FUNCTION "Sheet 4 (RSM)" : VOID	// FC 26
TITLE = Sheet 4 (RSM)
//HP FILM & TICM & TMAX (Analog)
AUTHOR : RJ
FAMILY : RSM
VERSION : 0.1
BEGIN
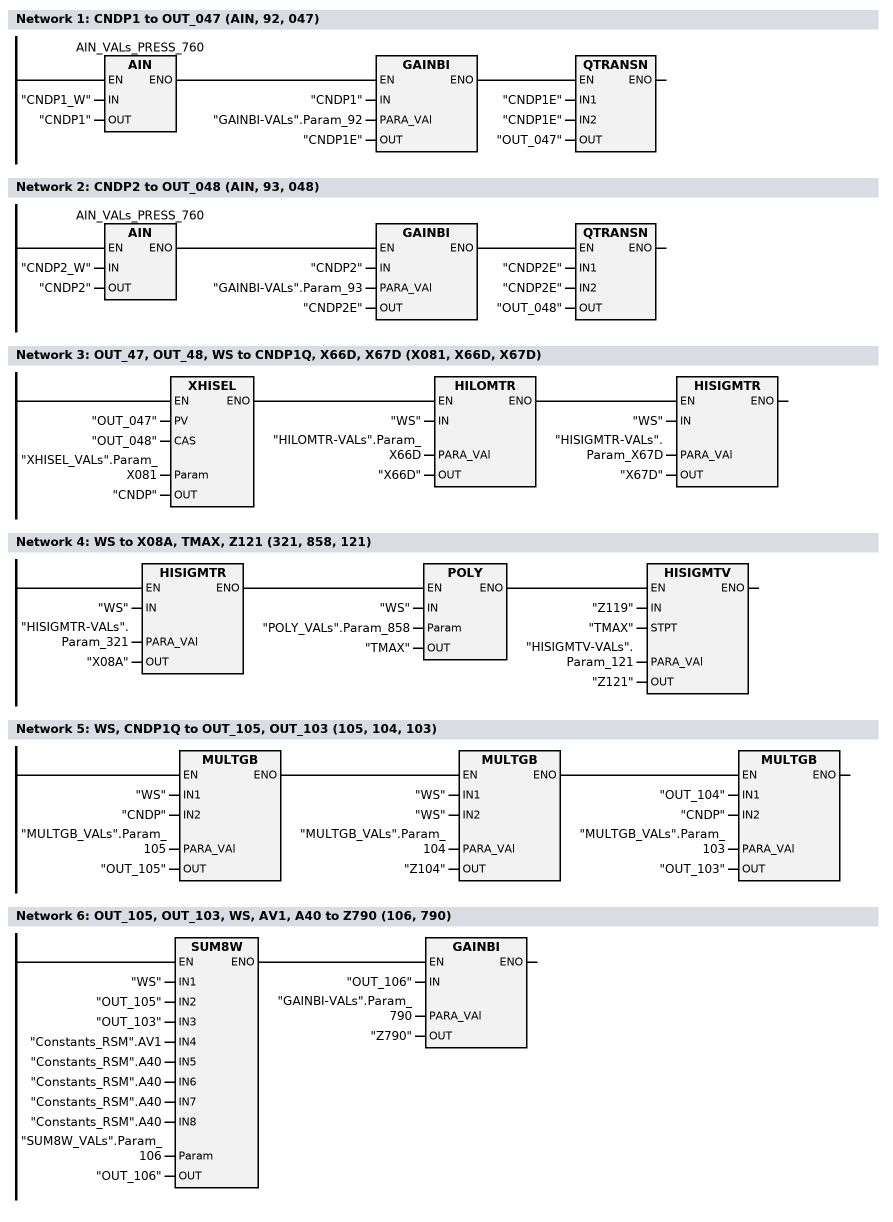
NETWORK
TITLE = CNDP1 to OUT_047 (AIN, 92, 047)
      A(;
      A(;
      CALL  "AIN" , "AIN_VALs_PRESS_760" (
           IN                       := "CNDP1_W",
           OUT                      := "CNDP1");
      A     BR;
      );
      JNB   _001;
      CALL  "GAINBI" (
           IN                       := "CNDP1",
           PARA_VAl                 := "GAINBI-VALs".Param_92,
           OUT                      := "CNDP1E");
_001: A     BR;
      );
      JNB   _002;
      CALL  "QTRANSN" (
           IN1                      := "CNDP1E",
           IN2                      := "CNDP1E",
           OUT                      := "OUT_047");
_002: NOP   0;
NETWORK
TITLE = CNDP2 to OUT_048 (AIN, 93, 048)
      A(;
      A(;
      CALL  "AIN" , "AIN_VALs_PRESS_760" (
           IN                       := "CNDP2_W",
           OUT                      := "CNDP2");
      A     BR;
      );
      JNB   _003;
      CALL  "GAINBI" (
           IN                       := "CNDP2",
           PARA_VAl                 := "GAINBI-VALs".Param_93,
           OUT                      := "CNDP2E");
_003: A     BR;
      );
      JNB   _004;
      CALL  "QTRANSN" (
           IN1                      := "CNDP2E",
           IN2                      := "CNDP2E",
           OUT                      := "OUT_048");
_004: NOP   0;
NETWORK
TITLE = OUT_47, OUT_48, WS to CNDP1Q, X66D, X67D (X081, X66D, X67D)
      A(;
      A(;
      CALL  "XHISEL" (
           PV                       := "OUT_047",
           CAS                      := "OUT_048",
           Param                    := "XHISEL_VALs".Param_X081,
           OUT                      := "CNDP");
      A     BR;
      );
      JNB   _005;
      CALL  "HILOMTR" (
           IN                       := "WS",
           PARA_VAl                 := "HILOMTR-VALs".Param_X66D,
           OUT                      := "X66D");
_005: A     BR;
      );
      JNB   _006;
      CALL  "HISIGMTR" (
           IN                       := "WS",
           PARA_VAl                 := "HISIGMTR-VALs".Param_X67D,
           OUT                      := "X67D");
_006: NOP   0;
NETWORK
TITLE = WS to X08A, TMAX, Z121 (321, 858, 121)
      A(;
      A(;
      CALL  "HISIGMTR" (
           IN                       := "WS",
           PARA_VAl                 := "HISIGMTR-VALs".Param_321,
           OUT                      := "X08A");
      A     BR;
      );
      JNB   _007;
      CALL  "POLY" (
           IN                       := "WS",
           Param                    := "POLY_VALs".Param_858,
           OUT                      := "TMAX");
_007: A     BR;
      );
      JNB   _008;
      CALL  "HISIGMTV" (
           IN                       := "Z119",
           STPT                     := "TMAX",
           PARA_VAl                 := "HISIGMTV-VALs".Param_121,
           OUT                      := "Z121");
_008: NOP   0;
NETWORK
TITLE = WS, CNDP1Q to OUT_105, OUT_103 (105, 104, 103)
      A(;
      A(;
      CALL  "MULTGB" (
           IN1                      := "WS",
           IN2                      := "CNDP",
           PARA_VAl                 := "MULTGB_VALs".Param_105,
           OUT                      := "OUT_105");
      A     BR;
      );
      JNB   _009;
      CALL  "MULTGB" (
           IN1                      := "WS",
           IN2                      := "WS",
           PARA_VAl                 := "MULTGB_VALs".Param_104,
           OUT                      := "Z104");
_009: A     BR;
      );
      JNB   _00a;
      CALL  "MULTGB" (
           IN1                      := "OUT_104",
           IN2                      := "CNDP",
           PARA_VAl                 := "MULTGB_VALs".Param_103,
           OUT                      := "OUT_103");
_00a: NOP   0;
NETWORK
TITLE = OUT_105, OUT_103, WS, AV1, A40 to Z790 (106, 790)
      A(;
      CALL  "SUM8W" (
           IN1                      := "WS",
           IN2                      := "OUT_105",
           IN3                      := "OUT_103",
           IN4                      := "Constants_RSM".AV1,
           IN5                      := "Constants_RSM".A40,
           IN6                      := "Constants_RSM".A40,
           IN7                      := "Constants_RSM".A40,
           IN8                      := "Constants_RSM".A40,
           Param                    := "SUM8W_VALs".Param_106,
           OUT                      := "OUT_106");
      A     BR;
      );
      JNB   _00b;
      CALL  "GAINBI" (
           IN                       := "OUT_106",
           PARA_VAl                 := "GAINBI-VALs".Param_790,
           OUT                      := "Z790");
_00b: NOP   0;
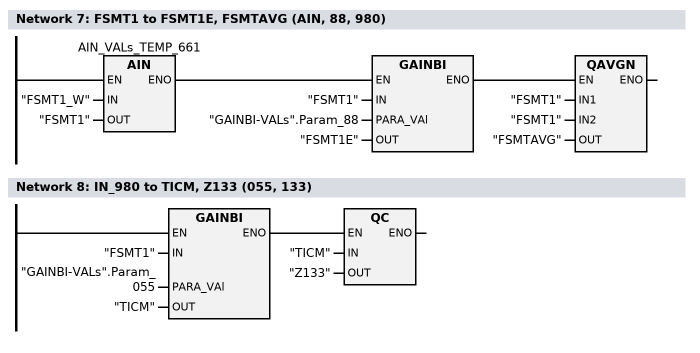
NETWORK
TITLE = FSMT1 to FSMT1E, FSMTAVG (AIN, 88, 980)
      A(;
      A(;
      CALL  "AIN" , "AIN_VALs_TEMP_661" (
           IN                       := "FSMT1_W",
           OUT                      := "FSMT1");
      A     BR;
      );
      JNB   _00c;
      CALL  "GAINBI" (
           IN                       := "FSMT1",
           PARA_VAl                 := "GAINBI-VALs".Param_88,
           OUT                      := "FSMT1E");
_00c: A     BR;
      );
      JNB   _00d;
      CALL  "QAVGN" (
           IN1                      := "FSMT1",
           IN2                      := "FSMT1",
           OUT                      := "FSMTAVG");
_00d: NOP   0;
NETWORK
TITLE = IN_980 to TICM, Z133 (055, 133)
      A(;
      CALL  "GAINBI" (
           IN                       := "FSMT1",
           PARA_VAl                 := "GAINBI-VALs".Param_055,
           OUT                      := "TICM");
      A     BR;
      );
      JNB   _00e;
      CALL  "QC" (
           IN                       := "TICM",
           OUT                      := "Z133");
_00e: NOP   0;
END_FUNCTION

FUNCTION "Sheet 5 (RSM)" : VOID	// FC 27
TITLE = Sheet 5 (RSM)
//MWINC LOGIC (Digital)
AUTHOR : RJ
FAMILY : RSM
VERSION : 0.1
BEGIN
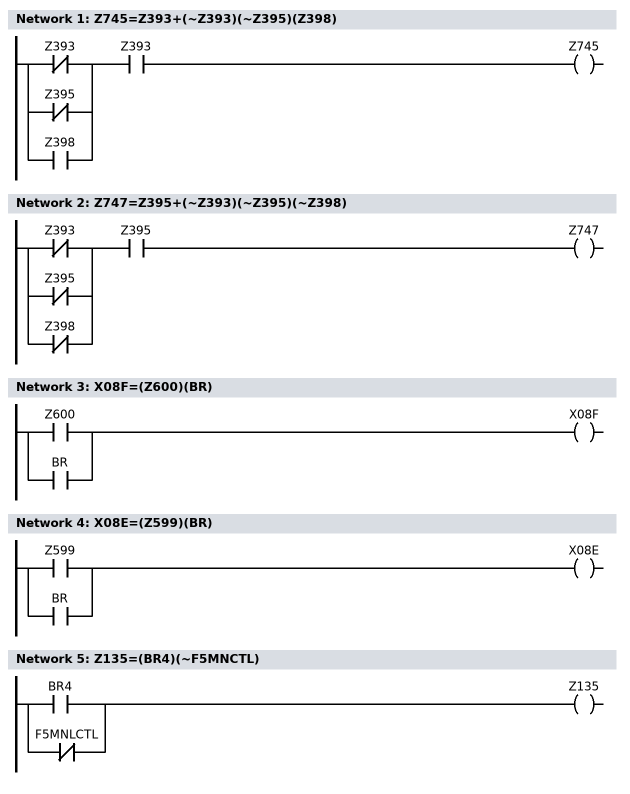
NETWORK
TITLE = Z745=Z393+(~Z393)(~Z395)(Z398)
      A(;
      ON    "Z393";
      ON    "Z395";
      O     "Z398";
      );
      A     "Z393";
      =     "Z745";
NETWORK
TITLE = Z747=Z395+(~Z393)(~Z395)(~Z398)
      A(;
      ON    "Z393";
      ON    "Z395";
      ON    "Z398";
      );
      A     "Z395";
      =     "Z747";
NETWORK
TITLE = X08F=(Z600)(BR)
      O     "Z600";
      O     "BR";
      =     "X08F";
NETWORK
TITLE = X08E=(Z599)(BR)
      O     "Z599";
      O     "BR";
      =     "X08E";
NETWORK
TITLE = Z135=(BR4)(~F5MNCTL)
      O     "BR4";
      ON    "F5MNLCTL";
      =     "Z135";
END_FUNCTION

FUNCTION "Sheet 7 (RSM)" : VOID	// FC 28
TITLE = Sheet 7 (RSM)
//HP INVALID LOGIC (Digital)
//
AUTHOR : RJ
FAMILY : RSM
VERSION : 0.1
BEGIN
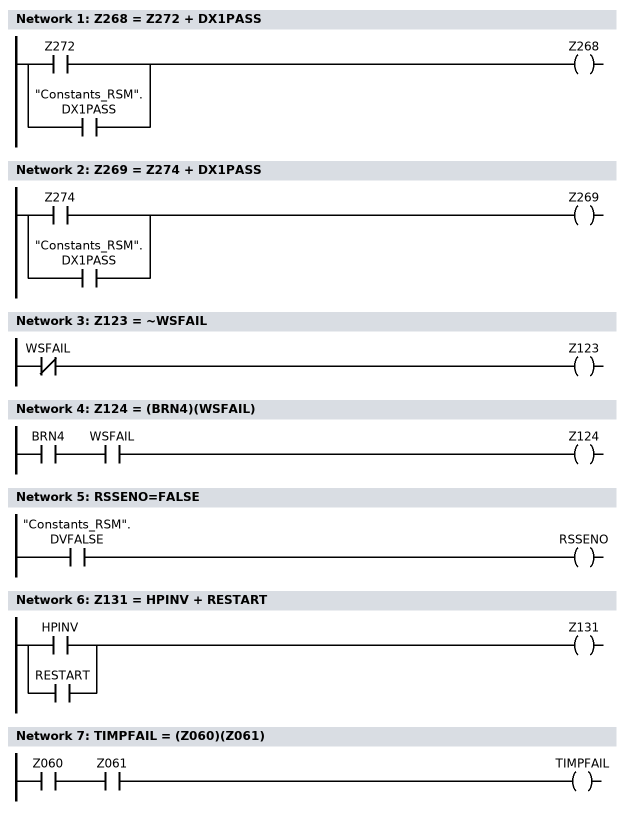
NETWORK
TITLE = Z268 = Z272 + DX1PASS
      O     "Z272";
      O     "Constants_RSM".DX1PASS;
      =     "Z268";
NETWORK
TITLE = Z269 = Z274 + DX1PASS
      O     "Z274";
      O     "Constants_RSM".DX1PASS;
      =     "Z269";
NETWORK
TITLE = Z123 = ~WSFAIL
      AN    "WSFAIL";
      =     "Z123";
NETWORK
TITLE = Z124 = (BRN4)(WSFAIL)
      A     "BRN4";
      A     "WSFAIL";
      =     "Z124";
NETWORK
TITLE = RSSENO=FALSE
      A     "Constants_RSM".DVFALSE;
      =     "RSSENO";
NETWORK
TITLE = Z131 = HPINV + RESTART
      O     "HPINV";
      O     "RESTART";
      =     "Z131";
NETWORK
TITLE = TIMPFAIL = (Z060)(Z061)
      A     "Z060";
      A     "Z061";
      =     "TIMPFAIL";
NETWORK
TITLE = RESTART Singnal logic
//RESTART=RTRSWSFL+DVFALSE+TIMPFAIL+(RESTART)(Z133)+(DX1PASS)(OUT_180)
      O     "RTRSWSFL";
      O     "Constants_RSM".DVFALSE;
      O     "TIMPFAIL";
      O;
      A     "Z133";
      A     "RESTART";
      O(;
      A     "Constants_RSM".DX1PASS;
      S     "OUT_180";
      A     "OUT_180";
      R     "OUT_180";
      A     "OUT_180";
      );
      =     "RESTART";
END_FUNCTION

FUNCTION "RESETSUM" : VOID	// FC 29
AUTHOR : RJ
VERSION : 0.0
VAR_INPUT
  FFLG : BOOL ;
  RSET : BOOL ;
  RUN : BOOL ;
  IN : REAL ;
  Param : STRUCT
   RCNT : REAL ;
   GAIN : REAL ;
   TRST : REAL ;
  END_STRUCT ;
END_VAR
VAR_IN_OUT
  OUT : REAL ;
END_VAR
VAR_TEMP
  TEMP : REAL ;
  RCNT : REAL ;
  GAIN : REAL ;
  TRST : REAL ;
END_VAR
BEGIN
// body was compiled from an SCL source; compiled code not shown
END_FUNCTION

FUNCTION "Sheet 6 (RSM)" : VOID	// FC 30
TITLE = Sheet 6 (RSM)
//HP Stress Counters (Analog)
AUTHOR : RJ
FAMILY : RSM
VERSION : 0.1
BEGIN
NETWORK
TITLE = AV1, DVFALSE, RESTART to X080, HPINV, HPICOL (129, 320, 130)
      A(;
      A(;
      A     "Constants_RSM".DVFALSE;
      =     L 0.0;
      BLD   103;
      A     "RESTART";
      =     L 0.1;
      BLD   103;
      A     "Z131";
      =     L 0.2;
      BLD   103;
      CALL  "RESETSUM" (
           FFLG                     := L 0.0,
           RSET                     := L 0.1,
           RUN                      := L 0.2,
           IN                       := "Constants_RSM".AV1,
           Param                    := "RESETSUM_VALs".Param_129,
           OUT                      := "HPICOL");
      A     BR;
      );
      JNB   _001;
      CALL  "HISIGMTR" (
           IN                       := "HPICOL",
           PARA_VAl                 := "HISIGMTR-VALs".Param_320,
           OUT                      := "X08D");
_001: A     BR;
      );
      JNB   _002;
      CALL  "LOSIGMTR" (
           IN                       := "HPICOL",
           PARA_VAl                 := "LOSIGMTR-VALs".Param_130,
           OUT                      := "HPINV");
_002: NOP   0;
NETWORK
TITLE = AV1, HPICOL to Z272 (270, 271, 272)
      A(;
      A     "Constants_RSM".DVFALSE;
      =     L 0.0;
      BLD   103;
      A     "Z272";
      =     L 0.1;
      BLD   103;
      A     "OUT_270";
      =     L 0.2;
      BLD   103;
      A(;
      CALL  "HISIGMTR" (
           IN                       := "HPICOL",
           PARA_VAl                 := "HISIGMTR-VALs".Param_270,
           OUT                      := "OUT_270");
      A     BR;
      );
      JNB   _003;
      CALL  "RESETSUM" (
           FFLG                     := L 0.0,
           RSET                     := L 0.1,
           RUN                      := L 0.2,
           IN                       := "Constants_RSM".AV1,
           Param                    := "RESETSUM_VALs".Param_271,
           OUT                      := "ONEMINCT");
_003: A     BR;
      );
      JNB   _004;
      CALL  "HISIGMTR" (
           IN                       := "ONEMINCT",
           PARA_VAl                 := "HISIGMTR-VALs".Param_272,
           OUT                      := "Z272");
_004: NOP   0;
NETWORK
TITLE = AV1, DVFALSE, DVTRUE to T5SEC (317, 318)
      A(;
      A     "Constants_RSM".DVFALSE;
      =     L 0.0;
      BLD   103;
      A     "T5SEC";
      =     L 0.1;
      BLD   103;
      A     "Constants_RSM".DVTRUE;
      =     L 0.2;
      BLD   103;
      CALL  "RESETSUM" (
           FFLG                     := L 0.0,
           RSET                     := L 0.1,
           RUN                      := L 0.2,
           IN                       := "Constants_RSM".AV1,
           Param                    := "RESETSUM_VALs".Param_317,
           OUT                      := "OUT_317");
      A     BR;
      );
      JNB   _005;
      CALL  "HISIGMTR" (
           IN                       := "OUT_317",
           PARA_VAl                 := "HISIGMTR-VALs".Param_318,
           OUT                      := "T5SEC");
_005: NOP   0;
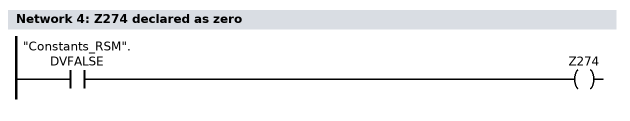
NETWORK
TITLE = Z274 declared as zero
      A     "Constants_RSM".DVFALSE;
      =     "Z274";
NETWORK
TITLE = AV1, Z123, Z124 to RTRSWSFL (125, 126)
      A(;
      A     "Constants_RSM".DVFALSE;
      =     L 0.0;
      BLD   103;
      A     "Z123";
      =     L 0.1;
      BLD   103;
      A     "Z124";
      =     L 0.2;
      BLD   103;
      CALL  "RESETSUM" (
           FFLG                     := L 0.0,
           RSET                     := L 0.1,
           RUN                      := L 0.2,
           IN                       := "Constants_RSM".AV1,
           Param                    := "RESETSUM_VALs".Param_136,
           OUT                      := "ISPOUTCT");
      A     BR;
      );
      JNB   _006;
      CALL  "HISIGMTR" (
           IN                       := "ISPOUTCT",
           PARA_VAl                 := "HISIGMTR-VALs".Param_137,
           OUT                      := "RTRSWSFL");
_006: NOP   0;
END_FUNCTION

FUNCTION "HISIGMTV" : VOID	// FC 31
AUTHOR : Sabeeh
VERSION : 0.0
VAR_INPUT
  IN : REAL ;
  STPT : REAL ;
  PARA_VAl : STRUCT
   DBAN : REAL ;
  END_STRUCT ;
END_VAR
VAR_OUTPUT
  OUT : BOOL ;
END_VAR
BEGIN
// body was compiled from an SCL source; compiled code not shown
END_FUNCTION

FUNCTION "LOSIGMTV" : VOID	// FC 32
AUTHOR : Sabeeh
VERSION : 0.0
VAR_INPUT
  IN1 : REAL ;
  STPT : REAL ;
  PARA_VAl : STRUCT
   DBAN : REAL ;
  END_STRUCT ;
END_VAR
VAR_OUTPUT
  FLAG : BOOL ;
END_VAR
BEGIN
// body was compiled from an SCL source; compiled code not shown
END_FUNCTION

FUNCTION "HISEL10" : VOID	// FC 33
AUTHOR : Sabeeh
VERSION : 0.0
VAR_INPUT
  IN1 : REAL ;
  IN2 : REAL ;
END_VAR
VAR_OUTPUT
  OUT : REAL ;
END_VAR
BEGIN
// body was compiled from an SCL source; compiled code not shown
END_FUNCTION

FUNCTION "XLIMIT" : VOID	// FC 34
AUTHOR : Sabeeh
VERSION : 0.0
VAR_INPUT
  CAS : REAL ;
  PARA_VAl : STRUCT
   GAIN : REAL  := 1.000000e+000;
   BIAS : REAL ;
   SCLTOP : REAL  := 1.000000e+002;
   SCLBTM : REAL  := -1.000000e+002;
  END_STRUCT ;
END_VAR
VAR_OUTPUT
  OUT : REAL ;
END_VAR
VAR_TEMP
  TEMP : REAL ;
END_VAR
BEGIN
// body was compiled from an SCL source; compiled code not shown
END_FUNCTION

FUNCTION "LOSEL10" : VOID	// FC 35
AUTHOR : Sabeeh
VERSION : 0.0
VAR_INPUT
  IN1 : REAL ;
  IN2 : REAL ;
END_VAR
VAR_OUTPUT
  OUT : REAL ;
END_VAR
BEGIN
// body was compiled from an SCL source; compiled code not shown
END_FUNCTION

FUNCTION "Sheet 9 (RSM)" : VOID	// FC 36
TITLE = Sheet 9 (RSM)
//HP ROTSURF, T1-5 & TP1-4 (Analog)
AUTHOR : RJ
FAMILY : RSM
VERSION : 0.1
BEGIN
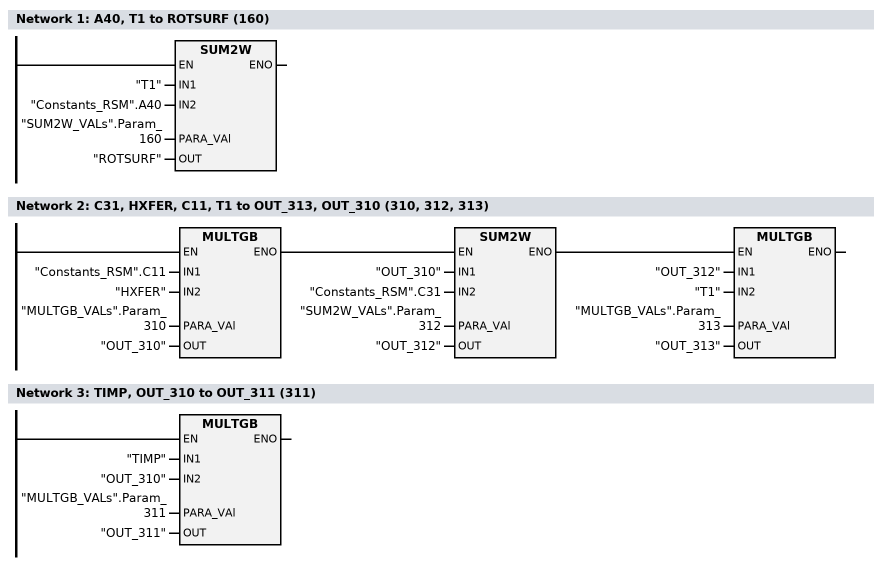
NETWORK
TITLE = A40, T1 to ROTSURF (160)
      CALL  "SUM2W" (
           IN1                      := "T1",
           IN2                      := "Constants_RSM".A40,
           PARA_VAl                 := "SUM2W_VALs".Param_160,
           OUT                      := "ROTSURF");
      NOP   0;
NETWORK
TITLE = C31, HXFER, C11, T1 to OUT_313, OUT_310 (310, 312, 313)
//IN1 of Block 312 should have a -ve weight w.r.f sheet 9 (RSM).
      A(;
      A(;
      CALL  "MULTGB" (
           IN1                      := "Constants_RSM".C11,
           IN2                      := "HXFER",
           PARA_VAl                 := "MULTGB_VALs".Param_310,
           OUT                      := "OUT_310");
      A     BR;
      );
      JNB   _001;
      CALL  "SUM2W" (
           IN1                      := "OUT_310",
           IN2                      := "Constants_RSM".C31,
           PARA_VAl                 := "SUM2W_VALs".Param_312,
           OUT                      := "OUT_312");
_001: A     BR;
      );
      JNB   _002;
      CALL  "MULTGB" (
           IN1                      := "OUT_312",
           IN2                      := "T1",
           PARA_VAl                 := "MULTGB_VALs".Param_313,
           OUT                      := "OUT_313");
_002: NOP   0;
NETWORK
TITLE = TIMP, OUT_310 to OUT_311 (311)
      CALL  "MULTGB" (
           IN1                      := "TIMP",
           IN2                      := "OUT_310",
           PARA_VAl                 := "MULTGB_VALs".Param_311,
           OUT                      := "OUT_311");
      NOP   0;
NETWORK
TITLE = Blocks 314, 315, 316
      A     "RESTART";
      =     L 0.0;
      BLD   103;
      A(;
      A     "T5SEC";
      =     L 0.1;
      BLD   103;
      A(;
      CALL  "SUM4W" (
           IN1                      := "OUT_311",
           IN2                      := "OUT_313",
           IN3                      := "T2",
           IN4                      := "Constants_RSM".A40,
           PARA_VAl                 := "SUM4W_VALs".Param_314,
           OUT                      := "TP1");
      A     BR;
      );
      JNB   _003;
      CALL  "TRANSF" (
           FLAG                     := L 0.1,
           IN1_y                    := "TP1",
           IN2_n                    := "T1",
           OUT                      := "OUT_315");
_003: A     BR;
      );
      JNB   _004;
      CALL  "TRANSF" (
           FLAG                     := L 0.0,
           IN1_y                    := "TICM",
           IN2_n                    := "OUT_315",
           OUT                      := "T1");
_004: NOP   0;
NETWORK
TITLE = Block 326, 327, 328
      A     "RESTART";
      =     L 0.0;
      BLD   103;
      A(;
      A     "T5SEC";
      =     L 0.1;
      BLD   103;
      A(;
      CALL  "SUM4W" (
           IN1                      := "T1",
           IN2                      := "T2",
           IN3                      := "T3",
           IN4                      := "Constants_RSM".A40,
           PARA_VAl                 := "SUM4W_VALs".Param_326,
           OUT                      := "TP2");
      A     BR;
      );
      JNB   _005;
      CALL  "TRANSF" (
           FLAG                     := L 0.1,
           IN1_y                    := "TP2",
           IN2_n                    := "T2",
           OUT                      := "OUT_327");
_005: A     BR;
      );
      JNB   _006;
      CALL  "TRANSF" (
           FLAG                     := L 0.0,
           IN1_y                    := "TICM",
           IN2_n                    := "OUT_327",
           OUT                      := "T2");
_006: NOP   0;
NETWORK
TITLE = Blocks 329, 330, 331
      A     "RESTART";
      =     L 0.0;
      BLD   103;
      A(;
      A     "T5SEC";
      =     L 0.1;
      BLD   103;
      A(;
      CALL  "SUM4W" (
           IN1                      := "T2",
           IN2                      := "T3",
           IN3                      := "T4",
           IN4                      := "Constants_RSM".A40,
           PARA_VAl                 := "SUM4W_VALs".Param_329,
           OUT                      := "TP3");
      A     BR;
      );
      JNB   _007;
      CALL  "TRANSF" (
           FLAG                     := L 0.1,
           IN1_y                    := "TP3",
           IN2_n                    := "T3",
           OUT                      := "OUT_330");
_007: A     BR;
      );
      JNB   _008;
      CALL  "TRANSF" (
           FLAG                     := L 0.0,
           IN1_y                    := "TICM",
           IN2_n                    := "OUT_330",
           OUT                      := "T3");
_008: NOP   0;
NETWORK
TITLE = Blocks 332, 333, 334
      A     "RESTART";
      =     L 0.0;
      BLD   103;
      A(;
      A     "T5SEC";
      =     L 0.1;
      BLD   103;
      A(;
      CALL  "SUM4W" (
           IN1                      := "T3",
           IN2                      := "T4",
           IN3                      := "T5",
           IN4                      := "Constants_RSM".A40,
           PARA_VAl                 := "SUM4W_VALs".Param_332,
           OUT                      := "TP4");
      A     BR;
      );
      JNB   _009;
      CALL  "TRANSF" (
           FLAG                     := L 0.1,
           IN1_y                    := "TP4",
           IN2_n                    := "T4",
           OUT                      := "OUT_333");
_009: A     BR;
      );
      JNB   _00a;
      CALL  "TRANSF" (
           FLAG                     := L 0.0,
           IN1_y                    := "TICM",
           IN2_n                    := "OUT_333",
           OUT                      := "T4");
_00a: NOP   0;
NETWORK
TITLE = Blocks 335, 336, 337
      A     "RESTART";
      =     L 0.0;
      BLD   103;
      A(;
      A     "T5SEC";
      =     L 0.1;
      BLD   103;
      A(;
      CALL  "SUM4W" (
           IN1                      := "T4",
           IN2                      := "T5",
           IN3                      := "T6",
           IN4                      := "Constants_RSM".A40,
           PARA_VAl                 := "SUM4W_VALs".Param_335,
           OUT                      := "TP5");
      A     BR;
      );
      JNB   _00b;
      CALL  "TRANSF" (
           FLAG                     := L 0.1,
           IN1_y                    := "TP5",
           IN2_n                    := "T5",
           OUT                      := "OUT_336");
_00b: A     BR;
      );
      JNB   _00c;
      CALL  "TRANSF" (
           FLAG                     := L 0.0,
           IN1_y                    := "TICM",
           IN2_n                    := "OUT_336",
           OUT                      := "T5");
_00c: NOP   0;
END_FUNCTION

FUNCTION "Sheet 8 (RSM)" : VOID	// FC 37
TITLE = Sheet 8 (RSM)
//HXFER & TWC (Analog)
AUTHOR : RJ
FAMILY : RSM
VERSION : 0.1
BEGIN
NETWORK
TITLE = Blocks 136, 137
      A(;
      A     "Constants_RSM".DVFALSE;
      =     L 0.0;
      BLD   103;
      A     "BRN4";
      =     L 0.1;
      BLD   103;
      A     "Z135";
      =     L 0.2;
      BLD   103;
      CALL  "RESETSUM" (
           FFLG                     := L 0.0,
           RSET                     := L 0.1,
           RUN                      := L 0.2,
           IN                       := "Constants_RSM".AV1,
           Param                    := P#DB30.DBX 60.0,
           OUT                      := "OUT_136");
      A     BR;
      );
      JNB   _001;
      CALL  "HISIGMTR" (
           IN                       := "OUT_136",
           PARA_VAl                 := "HISIGMTR-VALs".Param_221,
           OUT                      := "F5MNLCTL");
_001: NOP   0;
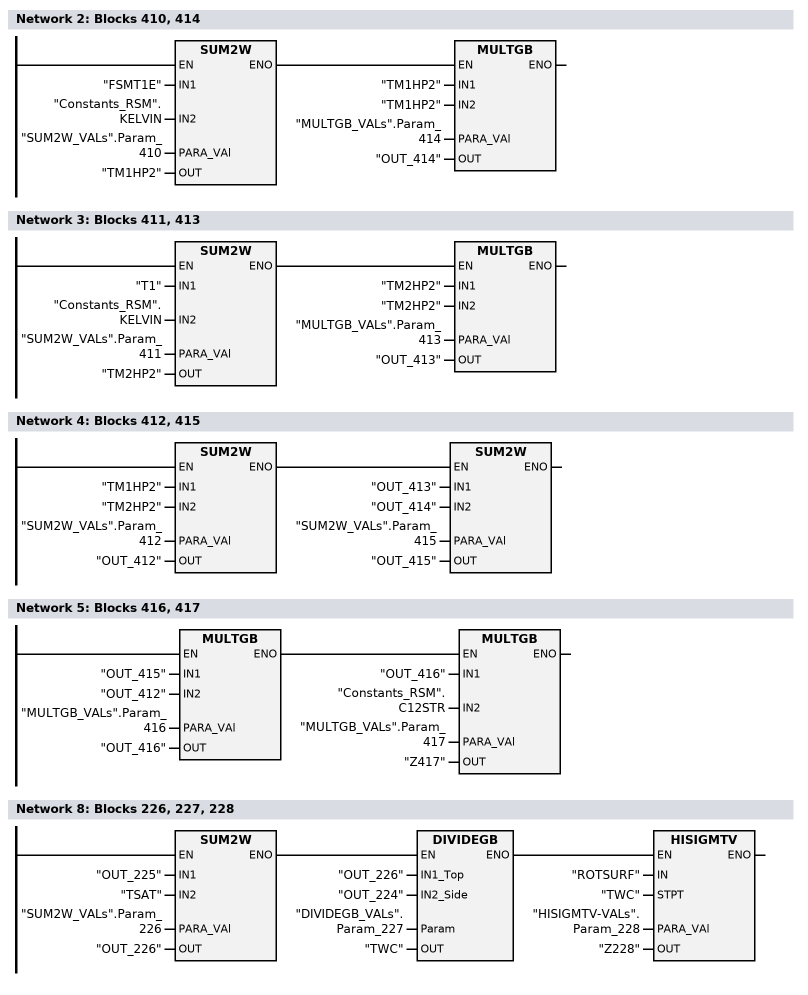
NETWORK
TITLE = Blocks 410, 414
      A(;
      CALL  "SUM2W" (
           IN1                      := "FSMT1E",
           IN2                      := "Constants_RSM".KELVIN,
           PARA_VAl                 := "SUM2W_VALs".Param_410,
           OUT                      := "TM1HP2");
      A     BR;
      );
      JNB   _002;
      CALL  "MULTGB" (
           IN1                      := "TM1HP2",
           IN2                      := "TM1HP2",
           PARA_VAl                 := "MULTGB_VALs".Param_414,
           OUT                      := "OUT_414");
_002: NOP   0;
NETWORK
TITLE = Blocks 411, 413
      A(;
      CALL  "SUM2W" (
           IN1                      := "T1",
           IN2                      := "Constants_RSM".KELVIN,
           PARA_VAl                 := "SUM2W_VALs".Param_411,
           OUT                      := "TM2HP2");
      A     BR;
      );
      JNB   _003;
      CALL  "MULTGB" (
           IN1                      := "TM2HP2",
           IN2                      := "TM2HP2",
           PARA_VAl                 := "MULTGB_VALs".Param_413,
           OUT                      := "OUT_413");
_003: NOP   0;
NETWORK
TITLE = Blocks 412, 415
      A(;
      CALL  "SUM2W" (
           IN1                      := "TM1HP2",
           IN2                      := "TM2HP2",
           PARA_VAl                 := "SUM2W_VALs".Param_412,
           OUT                      := "OUT_412");
      A     BR;
      );
      JNB   _004;
      CALL  "SUM2W" (
           IN1                      := "OUT_413",
           IN2                      := "OUT_414",
           PARA_VAl                 := "SUM2W_VALs".Param_415,
           OUT                      := "OUT_415");
_004: NOP   0;
NETWORK
TITLE = Blocks 416, 417
      A(;
      CALL  "MULTGB" (
           IN1                      := "OUT_415",
           IN2                      := "OUT_412",
           PARA_VAl                 := "MULTGB_VALs".Param_416,
           OUT                      := "OUT_416");
      A     BR;
      );
      JNB   _005;
      CALL  "MULTGB" (
           IN1                      := "OUT_416",
           IN2                      := "Constants_RSM".C12STR,
           PARA_VAl                 := "MULTGB_VALs".Param_417,
           OUT                      := "Z417");
_005: NOP   0;
NETWORK
TITLE = Blocks 122, 224, 221
      A(;
      A(;
      A     "XFER";
      =     L 0.0;
      BLD   103;
      CALL  "TRANSF" (
           FLAG                     := L 0.0,
           IN1_y                    := "Constants_RSM".C6,
           IN2_n                    := "Z790",
           OUT                      := "HXFER");
      A     BR;
      );
      JNB   _006;
      CALL  "GAINBI" (
           IN                       := "Z790",
           PARA_VAl                 := "GAINBI-VALs".Param_224,
           OUT                      := "OUT_224");
_006: A     BR;
      );
      JNB   _007;
      CALL  "HISIGMTR" (
           IN                       := "TMAX",
           PARA_VAl                 := "HISIGMTR-VALs".Param_X10G,
           OUT                      := "OUT_221");
_007: NOP   0;
NETWORK
TITLE = Blocks 222, 223, 225
      A(;
      A     "OUT_221";
      =     L 0.0;
      BLD   103;
      A(;
      CALL  "HISEL10" (
           IN1                      := "TMAX",
           IN2                      := "FSSTLO",
           OUT                      := "OUT_222");
      A     BR;
      );
      JNB   _008;
      CALL  "TRANSF" (
           FLAG                     := L 0.0,
           IN1_y                    := "OUT_222",
           IN2_n                    := "FSSTLO",
           OUT                      := "TSTM");
_008: A     BR;
      );
      JNB   _009;
      CALL  "MULTGB" (
           IN1                      := "Z790",
           IN2                      := "TSTM",
           PARA_VAl                 := "MULTGB_VALs".Param_225,
           OUT                      := "OUT_225");
_009: NOP   0;
NETWORK
TITLE = Blocks 226, 227, 228
      A(;
      A(;
      CALL  "SUM2W" (
           IN1                      := "OUT_225",
           IN2                      := "TSAT",
           PARA_VAl                 := "SUM2W_VALs".Param_226,
           OUT                      := "OUT_226");
      A     BR;
      );
      JNB   _00a;
      CALL  "DIVIDEGB" (
           IN1_Top                  := "OUT_226",
           IN2_Side                 := "OUT_224",
           Param                    := "DIVIDEGB_VALs".Param_227,
           OUT                      := "TWC");
_00a: A     BR;
      );
      JNB   _00b;
      CALL  "HISIGMTV" (
           IN                       := "ROTSURF",
           STPT                     := "TWC",
           PARA_VAl                 := "HISIGMTV-VALs".Param_228,
           OUT                      := "Z228");
_00b: NOP   0;
END_FUNCTION

FUNCTION "Sheet 10 (RSM)" : VOID	// FC 38
TITLE = Sheet 10 (RSM)
//HP TEMP T6-T15 (Analog)
AUTHOR : RJ
FAMILY : RSM
VERSION : 0.1
BEGIN
NETWORK
TITLE = Blocks 338, 339, 340
      A     "RESTART";
      =     L 0.0;
      BLD   103;
      A(;
      A     "T5SEC";
      =     L 0.1;
      BLD   103;
      A(;
      CALL  "SUM4W" (
           IN1                      := "T5",
           IN2                      := "T6",
           IN3                      := "T7",
           IN4                      := "Constants_RSM".A40,
           PARA_VAl                 := "SUM4W_VALs".Param_338,
           OUT                      := "TP6");
      A     BR;
      );
      JNB   _001;
      CALL  "TRANSF" (
           FLAG                     := L 0.1,
           IN1_y                    := "TP6",
           IN2_n                    := "T6",
           OUT                      := "OUT_339");
_001: A     BR;
      );
      JNB   _002;
      CALL  "TRANSF" (
           FLAG                     := L 0.0,
           IN1_y                    := "TICM",
           IN2_n                    := "OUT_339",
           OUT                      := "T6");
_002: NOP   0;
NETWORK
TITLE = Blocks 341, 342, 343
      A     "RESTART";
      =     L 0.0;
      BLD   103;
      A(;
      A     "T5SEC";
      =     L 0.1;
      BLD   103;
      A(;
      CALL  "SUM4W" (
           IN1                      := "T6",
           IN2                      := "T7",
           IN3                      := "T8",
           IN4                      := "Constants_RSM".A40,
           PARA_VAl                 := "SUM4W_VALs".Param_341,
           OUT                      := "TP7");
      A     BR;
      );
      JNB   _003;
      CALL  "TRANSF" (
           FLAG                     := L 0.1,
           IN1_y                    := "TP7",
           IN2_n                    := "T7",
           OUT                      := "OUT_342");
_003: A     BR;
      );
      JNB   _004;
      CALL  "TRANSF" (
           FLAG                     := L 0.0,
           IN1_y                    := "TICM",
           IN2_n                    := "OUT_342",
           OUT                      := "T7");
_004: NOP   0;
NETWORK
TITLE = Blocks 344, 345, 346
      A     "RESTART";
      =     L 0.0;
      BLD   103;
      A(;
      A     "T5SEC";
      =     L 0.1;
      BLD   103;
      A(;
      CALL  "SUM4W" (
           IN1                      := "T7",
           IN2                      := "T8",
           IN3                      := "T9",
           IN4                      := "Constants_RSM".A40,
           PARA_VAl                 := "SUM4W_VALs".Param_344,
           OUT                      := "TP8");
      A     BR;
      );
      JNB   _005;
      CALL  "TRANSF" (
           FLAG                     := L 0.1,
           IN1_y                    := "TP8",
           IN2_n                    := "T8",
           OUT                      := "OUT_345");
_005: A     BR;
      );
      JNB   _006;
      CALL  "TRANSF" (
           FLAG                     := L 0.0,
           IN1_y                    := "TICM",
           IN2_n                    := "OUT_345",
           OUT                      := "T8");
_006: NOP   0;
NETWORK
TITLE = Blocks 347, 348, 349
      A     "RESTART";
      =     L 0.0;
      BLD   103;
      A(;
      A     "T5SEC";
      =     L 0.1;
      BLD   103;
      A(;
      CALL  "SUM4W" (
           IN1                      := "T8",
           IN2                      := "T9",
           IN3                      := "T10",
           IN4                      := "Constants_RSM".A40,
           PARA_VAl                 := "SUM4W_VALs".Param_347,
           OUT                      := "TP9");
      A     BR;
      );
      JNB   _007;
      CALL  "TRANSF" (
           FLAG                     := L 0.1,
           IN1_y                    := "TP9",
           IN2_n                    := "T9",
           OUT                      := "OUT_348");
_007: A     BR;
      );
      JNB   _008;
      CALL  "TRANSF" (
           FLAG                     := L 0.0,
           IN1_y                    := "TICM",
           IN2_n                    := "OUT_348",
           OUT                      := "T9");
_008: NOP   0;
NETWORK
TITLE = Blocks 350, 351, 352
      A     "RESTART";
      =     L 0.0;
      BLD   103;
      A(;
      A     "T5SEC";
      =     L 0.1;
      BLD   103;
      A(;
      CALL  "SUM4W" (
           IN1                      := "T9",
           IN2                      := "T10",
           IN3                      := "T11",
           IN4                      := "Constants_RSM".A40,
           PARA_VAl                 := "SUM4W_VALs".Param_350,
           OUT                      := "TP10");
      A     BR;
      );
      JNB   _009;
      CALL  "TRANSF" (
           FLAG                     := L 0.1,
           IN1_y                    := "TP10",
           IN2_n                    := "T10",
           OUT                      := "OUT_351");
_009: A     BR;
      );
      JNB   _00a;
      CALL  "TRANSF" (
           FLAG                     := L 0.0,
           IN1_y                    := "TICM",
           IN2_n                    := "OUT_351",
           OUT                      := "T10");
_00a: NOP   0;
NETWORK
TITLE = Blocks 353, 354, 355
      A     "RESTART";
      =     L 0.0;
      BLD   103;
      A(;
      A     "T5SEC";
      =     L 0.1;
      BLD   103;
      A(;
      CALL  "SUM4W" (
           IN1                      := "T10",
           IN2                      := "T11",
           IN3                      := "T12",
           IN4                      := "Constants_RSM".A40,
           PARA_VAl                 := "SUM4W_VALs".Param_353,
           OUT                      := "TP11");
      A     BR;
      );
      JNB   _00b;
      CALL  "TRANSF" (
           FLAG                     := L 0.1,
           IN1_y                    := "TP11",
           IN2_n                    := "T11",
           OUT                      := "OUT_354");
_00b: A     BR;
      );
      JNB   _00c;
      CALL  "TRANSF" (
           FLAG                     := L 0.0,
           IN1_y                    := "TICM",
           IN2_n                    := "OUT_354",
           OUT                      := "T11");
_00c: NOP   0;
NETWORK
TITLE = Blocks 356, 357, 358
      A     "RESTART";
      =     L 0.0;
      BLD   103;
      A(;
      A     "T5SEC";
      =     L 0.1;
      BLD   103;
      A(;
      CALL  "SUM4W" (
           IN1                      := "T11",
           IN2                      := "T12",
           IN3                      := "T13",
           IN4                      := "Constants_RSM".A40,
           PARA_VAl                 := "SUM4W_VALs".Param_356,
           OUT                      := "TP12");
      A     BR;
      );
      JNB   _00d;
      CALL  "TRANSF" (
           FLAG                     := L 0.1,
           IN1_y                    := "TP12",
           IN2_n                    := "T12",
           OUT                      := "OUT_357");
_00d: A     BR;
      );
      JNB   _00e;
      CALL  "TRANSF" (
           FLAG                     := L 0.0,
           IN1_y                    := "TICM",
           IN2_n                    := "OUT_357",
           OUT                      := "T12");
_00e: NOP   0;
NETWORK
TITLE = Blocks 359, 360, 361
      A     "RESTART";
      =     L 0.0;
      BLD   103;
      A(;
      A     "T5SEC";
      =     L 0.1;
      BLD   103;
      A(;
      CALL  "SUM4W" (
           IN1                      := "T12",
           IN2                      := "T13",
           IN3                      := "T14",
           IN4                      := "Constants_RSM".A40,
           PARA_VAl                 := "SUM4W_VALs".Param_359,
           OUT                      := "TP12");
      A     BR;
      );
      JNB   _00f;
      CALL  "TRANSF" (
           FLAG                     := L 0.1,
           IN1_y                    := "TP12",
           IN2_n                    := "T12",
           OUT                      := "OUT_360");
_00f: A     BR;
      );
      JNB   _010;
      CALL  "TRANSF" (
           FLAG                     := L 0.0,
           IN1_y                    := "TICM",
           IN2_n                    := "OUT_360",
           OUT                      := "T12");
_010: NOP   0;
NETWORK
TITLE = Blocks 362, 363, 364
      A     "RESTART";
      =     L 0.0;
      BLD   103;
      A(;
      A     "T5SEC";
      =     L 0.1;
      BLD   103;
      A(;
      CALL  "SUM4W" (
           IN1                      := "T13",
           IN2                      := "T14",
           IN3                      := "T15",
           IN4                      := "Constants_RSM".A40,
           PARA_VAl                 := "SUM4W_VALs".Param_362,
           OUT                      := "TP14");
      A     BR;
      );
      JNB   _011;
      CALL  "TRANSF" (
           FLAG                     := L 0.1,
           IN1_y                    := "TP14",
           IN2_n                    := "T14",
           OUT                      := "OUT_363");
_011: A     BR;
      );
      JNB   _012;
      CALL  "TRANSF" (
           FLAG                     := L 0.0,
           IN1_y                    := "TICM",
           IN2_n                    := "OUT_363",
           OUT                      := "T14");
_012: NOP   0;
NETWORK
TITLE = Blocks 376, 377, 378
      A     "RESTART";
      =     L 0.0;
      BLD   103;
      A(;
      A     "T5SEC";
      =     L 0.1;
      BLD   103;
      A(;
      CALL  "SUM4W" (
           IN1                      := "T14",
           IN2                      := "T15",
           IN3                      := "T16",
           IN4                      := "Constants_RSM".A40,
           PARA_VAl                 := "SUM4W_VALs".Param_376,
           OUT                      := "TP15");
      A     BR;
      );
      JNB   _013;
      CALL  "TRANSF" (
           FLAG                     := L 0.1,
           IN1_y                    := "TP15",
           IN2_n                    := "T15",
           OUT                      := "OUT_377");
_013: A     BR;
      );
      JNB   _014;
      CALL  "TRANSF" (
           FLAG                     := L 0.0,
           IN1_y                    := "TICM",
           IN2_n                    := "OUT_377",
           OUT                      := "T15");
_014: NOP   0;
END_FUNCTION

FUNCTION "Sheet11 (RSM)" : VOID	// FC 39
TITLE = Sheet 11 (RSM)
//HP TEMP T16-T23 (Analog)
AUTHOR : RJ
FAMILY : RSM
VERSION : 0.1
BEGIN
NETWORK
TITLE = Blocks 301, 302, 303
      A     "RESTART";
      =     L 0.0;
      BLD   103;
      A(;
      A     "T5SEC";
      =     L 0.1;
      BLD   103;
      A(;
      CALL  "SUM4W" (
           IN1                      := "T15",
           IN2                      := "T16",
           IN3                      := "T17",
           IN4                      := "Constants_RSM".A40,
           PARA_VAl                 := "SUM4W_VALs".Param_301,
           OUT                      := "TP16");
      A     BR;
      );
      JNB   _001;
      CALL  "TRANSF" (
           FLAG                     := L 0.1,
           IN1_y                    := "TP16",
           IN2_n                    := "T16",
           OUT                      := "OUT_302");
_001: A     BR;
      );
      JNB   _002;
      CALL  "TRANSF" (
           FLAG                     := L 0.0,
           IN1_y                    := "TICM",
           IN2_n                    := "OUT_302",
           OUT                      := "T16");
_002: NOP   0;
NETWORK
TITLE = Block 304, 305, 306
      A     "RESTART";
      =     L 0.0;
      BLD   103;
      A(;
      A     "T5SEC";
      =     L 0.1;
      BLD   103;
      A(;
      CALL  "SUM4W" (
           IN1                      := "T16",
           IN2                      := "T17",
           IN3                      := "T18",
           IN4                      := "Constants_RSM".A40,
           PARA_VAl                 := "SUM4W_VALs".Param_304,
           OUT                      := "TP17");
      A     BR;
      );
      JNB   _003;
      CALL  "TRANSF" (
           FLAG                     := L 0.1,
           IN1_y                    := "TP17",
           IN2_n                    := "T17",
           OUT                      := "OUT_305");
_003: A     BR;
      );
      JNB   _004;
      CALL  "TRANSF" (
           FLAG                     := L 0.0,
           IN1_y                    := "TICM",
           IN2_n                    := "OUT_305",
           OUT                      := "T17");
_004: NOP   0;
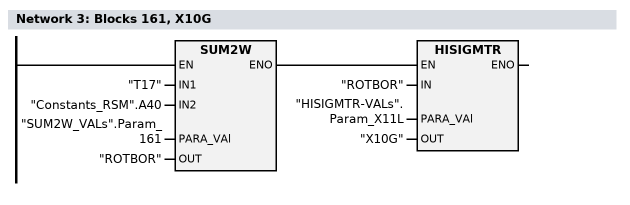
NETWORK
TITLE = Blocks 161, X10G
      A(;
      CALL  "SUM2W" (
           IN1                      := "T17",
           IN2                      := "Constants_RSM".A40,
           PARA_VAl                 := "SUM2W_VALs".Param_161,
           OUT                      := "ROTBOR");
      A     BR;
      );
      JNB   _005;
      CALL  "HISIGMTR" (
           IN                       := "ROTBOR",
           PARA_VAl                 := "HISIGMTR-VALs".Param_X11L,
           OUT                      := "X10G");
_005: NOP   0;
END_FUNCTION

FUNCTION "MULTGB" : VOID	// FC 40
AUTHOR : Sabeeh
VERSION : 0.0
VAR_INPUT
  IN1 : REAL ;
  IN2 : REAL ;
  PARA_VAl : STRUCT
   GAIN : REAL ;
   BIAS : REAL ;
  END_STRUCT ;
END_VAR
VAR_OUTPUT
  OUT : REAL ;
END_VAR
BEGIN
// body was compiled from an SCL source; compiled code not shown
END_FUNCTION

FUNCTION "SUM2W" : VOID	// FC 41
AUTHOR : Sabeeh
VERSION : 0.0
VAR_INPUT
  IN1 : REAL ;
  IN2 : REAL ;
  PARA_VAl : STRUCT
   WT1 : REAL ;
   WT2 : REAL ;
  END_STRUCT ;
END_VAR
VAR_OUTPUT
  OUT : REAL ;
END_VAR
BEGIN
// body was compiled from an SCL source; compiled code not shown
END_FUNCTION

FUNCTION "RATEMTR" : VOID	// FC 42
AUTHOR : RJ
VERSION : 0.0
VAR_INPUT
  IN : REAL ;
END_VAR
VAR_OUTPUT
  OUT : BOOL ;
END_VAR
VAR_IN_OUT
  Param : STRUCT
   OLDIN : REAL ;
   OLDT : TIME ;
   i : INT ;
   PRATE : REAL ;
   NRATE : REAL ;
   PDB : REAL ;
   NDB : REAL ;
  END_STRUCT ;
END_VAR
VAR_TEMP
  RATE : REAL ;
  NEWT : TIME ;
  TIME_ELAPSED : REAL ;
  OLDIN : REAL ;
  OLDT : TIME ;
  i : INT ;
  PRATE : REAL ;
  NRATE : REAL ;
  PDB : REAL ;
  NDB : REAL ;
END_VAR
BEGIN
// body was compiled from an SCL source; compiled code not shown
END_FUNCTION

FUNCTION "XSUM" : VOID	// FC 43
AUTHOR : Sabeeh
VERSION : 0.0
VAR_INPUT
  PV : REAL ;
  CAS : REAL ;
  PARA_VAl : STRUCT
   PVGAIN : REAL ;
   PVBIAS : REAL ;
   CASGAIN : REAL ;
   CASBIAS : REAL ;
   SCALETOP : REAL ;
   SCALEBOT : REAL ;
  END_STRUCT ;
END_VAR
VAR_OUTPUT
  OUTPUT : REAL ;
END_VAR
VAR_TEMP
  PVGB : REAL ;
  CASGB : REAL ;
END_VAR
BEGIN
// body was compiled from an SCL source; compiled code not shown
END_FUNCTION

FUNCTION "XTRANSF" : VOID	// FC 44
AUTHOR : Sabeeh
VERSION : 0.0
VAR_INPUT
  PV_Y : REAL ;
  CAS_N : REAL ;
  FLAG : BOOL ;
  PARA_VAl : STRUCT
   PV_YGAIN : REAL ;
   PV_YBIAS : REAL ;
   CAS_NGAIN : REAL ;
   CAS_NBIAS : REAL ;
   SCALETOP : REAL ;
   SCALEBOT : REAL ;
  END_STRUCT ;
END_VAR
VAR_OUTPUT
  OUTPUT : REAL ;
END_VAR
BEGIN
// body was compiled from an SCL source; compiled code not shown
END_FUNCTION

FUNCTION "Sheet 12 (RSM)" : VOID	// FC 45
TITLE = Sheet 12 (RSM)
//HP TAVG (Analog)
AUTHOR : RJ
FAMILY : RSM
VERSION : 0.1
BEGIN
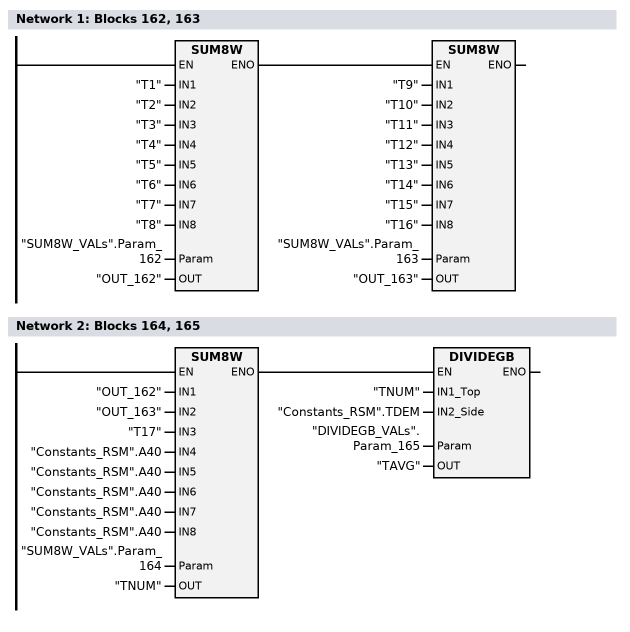
NETWORK
TITLE = Blocks 162, 163
      A(;
      CALL  "SUM8W" (
           IN1                      := "T1",
           IN2                      := "T2",
           IN3                      := "T3",
           IN4                      := "T4",
           IN5                      := "T5",
           IN6                      := "T6",
           IN7                      := "T7",
           IN8                      := "T8",
           Param                    := "SUM8W_VALs".Param_162,
           OUT                      := "OUT_162");
      A     BR;
      );
      JNB   _001;
      CALL  "SUM8W" (
           IN1                      := "T9",
           IN2                      := "T10",
           IN3                      := "T11",
           IN4                      := "T12",
           IN5                      := "T13",
           IN6                      := "T14",
           IN7                      := "T15",
           IN8                      := "T16",
           Param                    := "SUM8W_VALs".Param_163,
           OUT                      := "OUT_163");
_001: NOP   0;
NETWORK
TITLE = Blocks 164, 165
      A(;
      CALL  "SUM8W" (
           IN1                      := "OUT_162",
           IN2                      := "OUT_163",
           IN3                      := "T17",
           IN4                      := "Constants_RSM".A40,
           IN5                      := "Constants_RSM".A40,
           IN6                      := "Constants_RSM".A40,
           IN7                      := "Constants_RSM".A40,
           IN8                      := "Constants_RSM".A40,
           Param                    := "SUM8W_VALs".Param_164,
           OUT                      := "TNUM");
      A     BR;
      );
      JNB   _002;
      CALL  "DIVIDEGB" (
           IN1_Top                  := "TNUM",
           IN2_Side                 := "Constants_RSM".TDEM,
           Param                    := "DIVIDEGB_VALs".Param_165,
           OUT                      := "TAVG");
_002: NOP   0;
END_FUNCTION

FUNCTION "Sheet 13 (RSM)" : VOID	// FC 46
TITLE = Sheet 13 (RSM)
//HP EFFECTIVE TEMP DIFF. (Analog)
AUTHOR : RJ
FAMILY : RSM
VERSION : 0.1
BEGIN
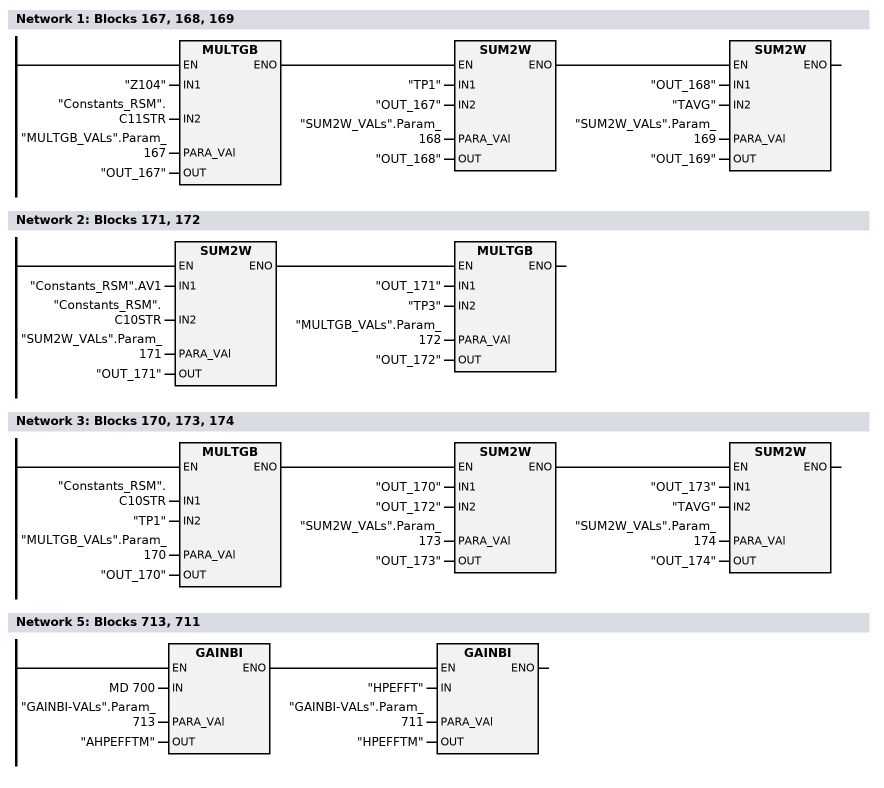
NETWORK
TITLE = Blocks 167, 168, 169
//IN2 of blocks 168 and 169 should have -ve weight. 
      A(;
      A(;
      CALL  "MULTGB" (
           IN1                      := "Z104",
           IN2                      := "Constants_RSM".C11STR,
           PARA_VAl                 := "MULTGB_VALs".Param_167,
           OUT                      := "OUT_167");
      A     BR;
      );
      JNB   _001;
      CALL  "SUM2W" (
           IN1                      := "TP1",
           IN2                      := "OUT_167",
           PARA_VAl                 := "SUM2W_VALs".Param_168,
           OUT                      := "OUT_168");
_001: A     BR;
      );
      JNB   _002;
      CALL  "SUM2W" (
           IN1                      := "OUT_168",
           IN2                      := "TAVG",
           PARA_VAl                 := "SUM2W_VALs".Param_169,
           OUT                      := "OUT_169");
_002: NOP   0;
NETWORK
TITLE = Blocks 171, 172
//IN2 of block 171 should have -ve weight.
      A(;
      CALL  "SUM2W" (
           IN1                      := "Constants_RSM".AV1,
           IN2                      := "Constants_RSM".C10STR,
           PARA_VAl                 := "SUM2W_VALs".Param_171,
           OUT                      := "OUT_171");
      A     BR;
      );
      JNB   _003;
      CALL  "MULTGB" (
           IN1                      := "OUT_171",
           IN2                      := "TP3",
           PARA_VAl                 := "MULTGB_VALs".Param_172,
           OUT                      := "OUT_172");
_003: NOP   0;
NETWORK
TITLE = Blocks 170, 173, 174
//IN2 of block 174 should have -ve weight.
      A(;
      A(;
      CALL  "MULTGB" (
           IN1                      := "Constants_RSM".C10STR,
           IN2                      := "TP1",
           PARA_VAl                 := "MULTGB_VALs".Param_170,
           OUT                      := "OUT_170");
      A     BR;
      );
      JNB   _004;
      CALL  "SUM2W" (
           IN1                      := "OUT_170",
           IN2                      := "OUT_172",
           PARA_VAl                 := "SUM2W_VALs".Param_173,
           OUT                      := "OUT_173");
_004: A     BR;
      );
      JNB   _005;
      CALL  "SUM2W" (
           IN1                      := "OUT_173",
           IN2                      := "TAVG",
           PARA_VAl                 := "SUM2W_VALs".Param_174,
           OUT                      := "OUT_174");
_005: NOP   0;
NETWORK
TITLE = Blocks 175, 185
      A(;
      A     "TROOTHP";
      =     L 0.0;
      BLD   103;
      CALL  "TRANSF" (
           FLAG                     := L 0.0,
           IN1_y                    := "OUT_174",
           IN2_n                    := "OUT_169",
           OUT                      := "HPEFFT");
      A     BR;
      );
      JNB   _006;
      L     "HPEFFT";
      ABS;
      T     "AHPEFFT";
_006: NOP   0;
NETWORK
TITLE = Blocks 713, 711
      A(;
      CALL  "GAINBI" (
           IN                       := MD 700,
           PARA_VAl                 := "GAINBI-VALs".Param_713,
           OUT                      := "AHPEFFTM");
      A     BR;
      );
      JNB   _007;
      CALL  "GAINBI" (
           IN                       := "HPEFFT",
           PARA_VAl                 := "GAINBI-VALs".Param_711,
           OUT                      := "HPEFFTM");
_007: NOP   0;
END_FUNCTION

FUNCTION "Sheet 14 (RSM)" : VOID	// FC 47
TITLE = Sheet 14 (RSM)
//All variables declared as zero
AUTHOR : RJ
FAMILY : RSM
VERSION : 0.1
BEGIN
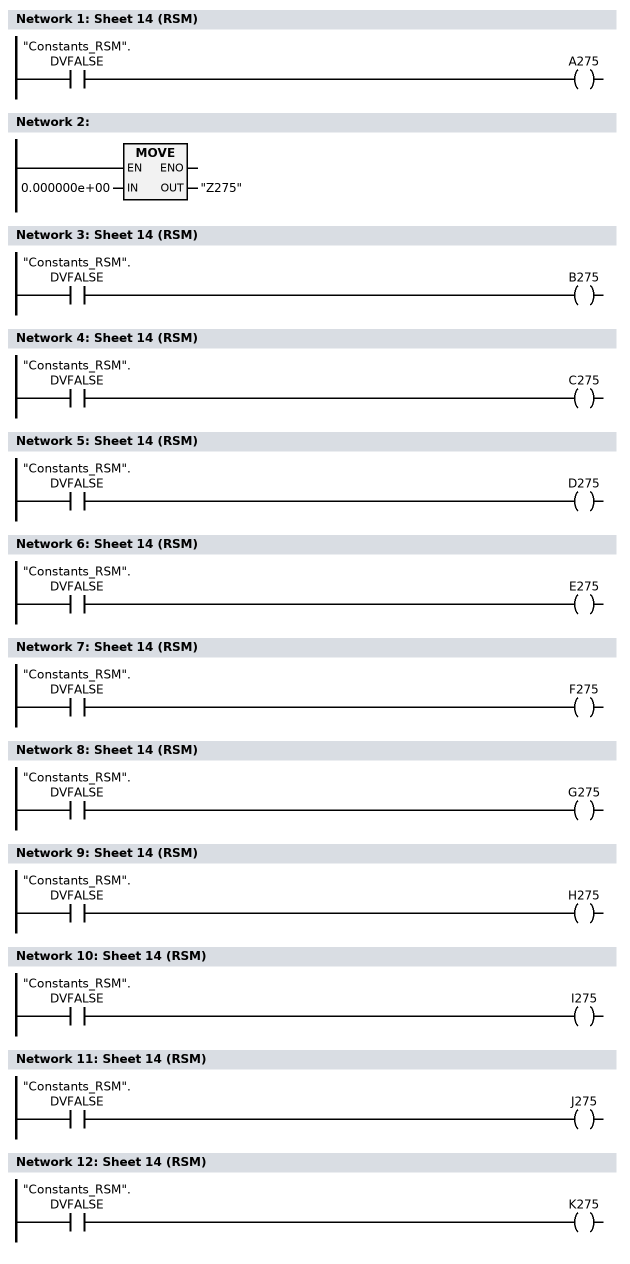
NETWORK
TITLE = Sheet 14 (RSM)
      A     "Constants_RSM".DVFALSE;
      =     "A275";
NETWORK
TITLE =
      L     0.000000e+00;
      T     "Z275";
      NOP   0;
NETWORK
TITLE = Sheet 14 (RSM)
      A     "Constants_RSM".DVFALSE;
      =     "B275";
NETWORK
TITLE = Sheet 14 (RSM)
      A     "Constants_RSM".DVFALSE;
      =     "C275";
NETWORK
TITLE = Sheet 14 (RSM)
      A     "Constants_RSM".DVFALSE;
      =     "D275";
NETWORK
TITLE = Sheet 14 (RSM)
      A     "Constants_RSM".DVFALSE;
      =     "E275";
NETWORK
TITLE = Sheet 14 (RSM)
      A     "Constants_RSM".DVFALSE;
      =     "F275";
NETWORK
TITLE = Sheet 14 (RSM)
      A     "Constants_RSM".DVFALSE;
      =     "G275";
NETWORK
TITLE = Sheet 14 (RSM)
      A     "Constants_RSM".DVFALSE;
      =     "H275";
NETWORK
TITLE = Sheet 14 (RSM)
      A     "Constants_RSM".DVFALSE;
      =     "I275";
NETWORK
TITLE = Sheet 14 (RSM)
      A     "Constants_RSM".DVFALSE;
      =     "J275";
NETWORK
TITLE = Sheet 14 (RSM)
      A     "Constants_RSM".DVFALSE;
      =     "K275";
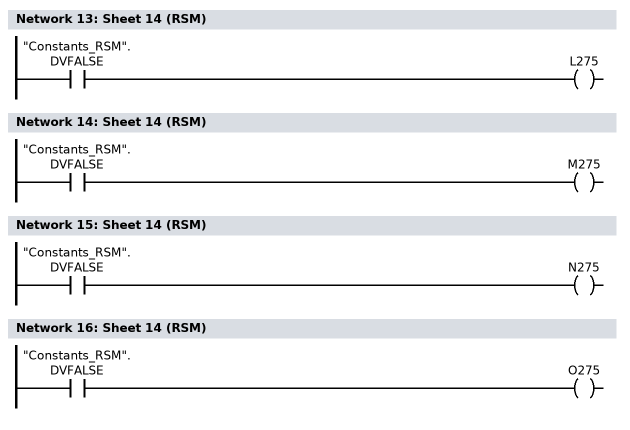
NETWORK
TITLE = Sheet 14 (RSM)
      A     "Constants_RSM".DVFALSE;
      =     "L275";
NETWORK
TITLE = Sheet 14 (RSM)
      A     "Constants_RSM".DVFALSE;
      =     "M275";
NETWORK
TITLE = Sheet 14 (RSM)
      A     "Constants_RSM".DVFALSE;
      =     "N275";
NETWORK
TITLE = Sheet 14 (RSM)
      A     "Constants_RSM".DVFALSE;
      =     "O275";
END_FUNCTION

FUNCTION "Sheet 15 (RSM)" : VOID	// FC 48
TITLE = Sheet 15 (RSM)
//HP TD1FT1-15 (Analog)
AUTHOR : RJ
FAMILY : RSM
VERSION : 0.1
BEGIN
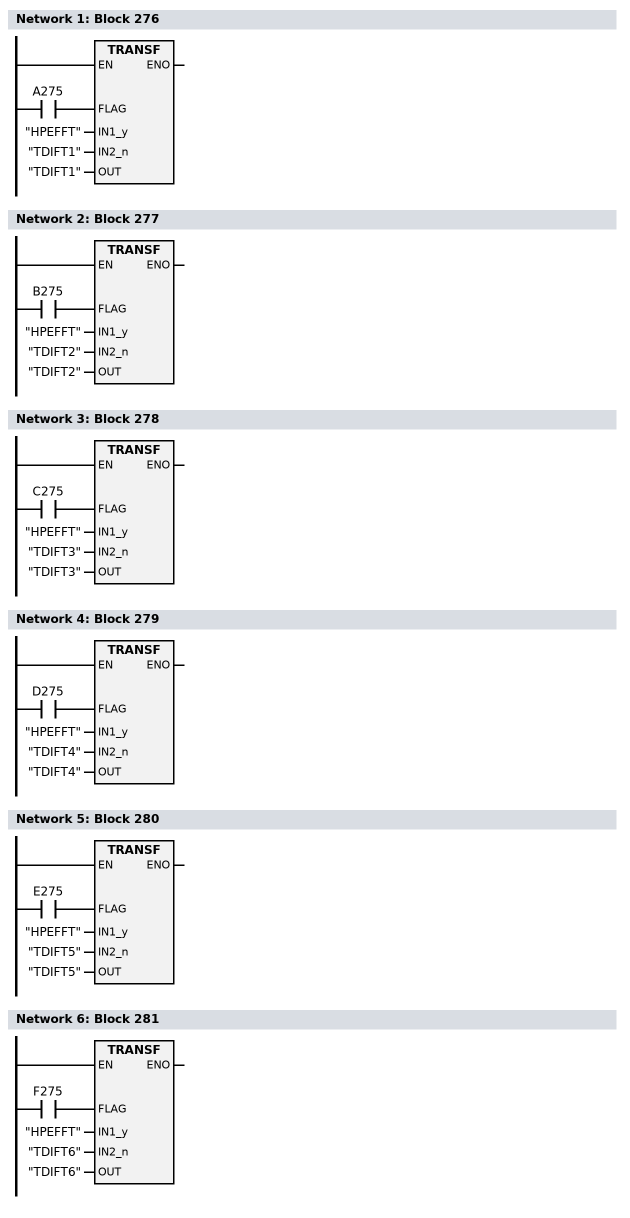
NETWORK
TITLE = Block 276
      A     "A275";
      =     L 0.0;
      BLD   103;
      CALL  "TRANSF" (
           FLAG                     := L 0.0,
           IN1_y                    := "HPEFFT",
           IN2_n                    := "TDIFT1",
           OUT                      := "TDIFT1");
      NOP   0;
NETWORK
TITLE = Block 277
      A     "B275";
      =     L 0.0;
      BLD   103;
      CALL  "TRANSF" (
           FLAG                     := L 0.0,
           IN1_y                    := "HPEFFT",
           IN2_n                    := "TDIFT2",
           OUT                      := "TDIFT2");
      NOP   0;
NETWORK
TITLE = Block 278
      A     "C275";
      =     L 0.0;
      BLD   103;
      CALL  "TRANSF" (
           FLAG                     := L 0.0,
           IN1_y                    := "HPEFFT",
           IN2_n                    := "TDIFT3",
           OUT                      := "TDIFT3");
      NOP   0;
NETWORK
TITLE = Block 279
      A     "D275";
      =     L 0.0;
      BLD   103;
      CALL  "TRANSF" (
           FLAG                     := L 0.0,
           IN1_y                    := "HPEFFT",
           IN2_n                    := "TDIFT4",
           OUT                      := "TDIFT4");
      NOP   0;
NETWORK
TITLE = Block 280
      A     "E275";
      =     L 0.0;
      BLD   103;
      CALL  "TRANSF" (
           FLAG                     := L 0.0,
           IN1_y                    := "HPEFFT",
           IN2_n                    := "TDIFT5",
           OUT                      := "TDIFT5");
      NOP   0;
NETWORK
TITLE = Block 281
      A     "F275";
      =     L 0.0;
      BLD   103;
      CALL  "TRANSF" (
           FLAG                     := L 0.0,
           IN1_y                    := "HPEFFT",
           IN2_n                    := "TDIFT6",
           OUT                      := "TDIFT6");
      NOP   0;
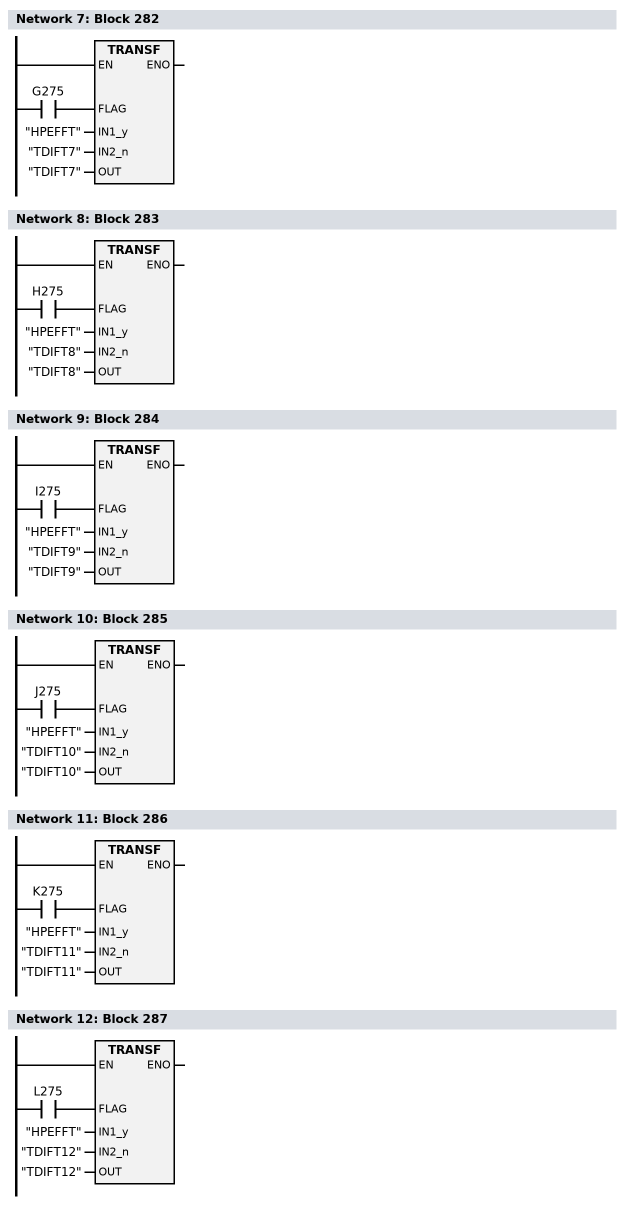
NETWORK
TITLE = Block 282
      A     "G275";
      =     L 0.0;
      BLD   103;
      CALL  "TRANSF" (
           FLAG                     := L 0.0,
           IN1_y                    := "HPEFFT",
           IN2_n                    := "TDIFT7",
           OUT                      := "TDIFT7");
      NOP   0;
NETWORK
TITLE = Block 283
      A     "H275";
      =     L 0.0;
      BLD   103;
      CALL  "TRANSF" (
           FLAG                     := L 0.0,
           IN1_y                    := "HPEFFT",
           IN2_n                    := "TDIFT8",
           OUT                      := "TDIFT8");
      NOP   0;
NETWORK
TITLE = Block 284
      A     "I275";
      =     L 0.0;
      BLD   103;
      CALL  "TRANSF" (
           FLAG                     := L 0.0,
           IN1_y                    := "HPEFFT",
           IN2_n                    := "TDIFT9",
           OUT                      := "TDIFT9");
      NOP   0;
NETWORK
TITLE = Block 285
      A     "J275";
      =     L 0.0;
      BLD   103;
      CALL  "TRANSF" (
           FLAG                     := L 0.0,
           IN1_y                    := "HPEFFT",
           IN2_n                    := "TDIFT10",
           OUT                      := "TDIFT10");
      NOP   0;
NETWORK
TITLE = Block 286
      A     "K275";
      =     L 0.0;
      BLD   103;
      CALL  "TRANSF" (
           FLAG                     := L 0.0,
           IN1_y                    := "HPEFFT",
           IN2_n                    := "TDIFT11",
           OUT                      := "TDIFT11");
      NOP   0;
NETWORK
TITLE = Block 287
      A     "L275";
      =     L 0.0;
      BLD   103;
      CALL  "TRANSF" (
           FLAG                     := L 0.0,
           IN1_y                    := "HPEFFT",
           IN2_n                    := "TDIFT12",
           OUT                      := "TDIFT12");
      NOP   0;
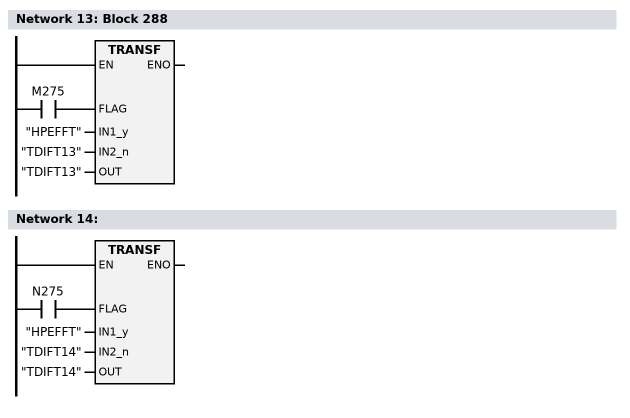
NETWORK
TITLE = Block 288
      A     "M275";
      =     L 0.0;
      BLD   103;
      CALL  "TRANSF" (
           FLAG                     := L 0.0,
           IN1_y                    := "HPEFFT",
           IN2_n                    := "TDIFT13",
           OUT                      := "TDIFT13");
      NOP   0;
NETWORK
TITLE =
      A     "N275";
      =     L 0.0;
      BLD   103;
      CALL  "TRANSF" (
           FLAG                     := L 0.0,
           IN1_y                    := "HPEFFT",
           IN2_n                    := "TDIFT14",
           OUT                      := "TDIFT14");
      NOP   0;
END_FUNCTION

FUNCTION "Sheet 16 (RSM)" : VOID	// FC 51
TITLE = Sheet 16 (RSM)
//HP ANTIC. DIFF. (Analog)
AUTHOR : RJ
FAMILY : RSM
VERSION : 0.1
BEGIN
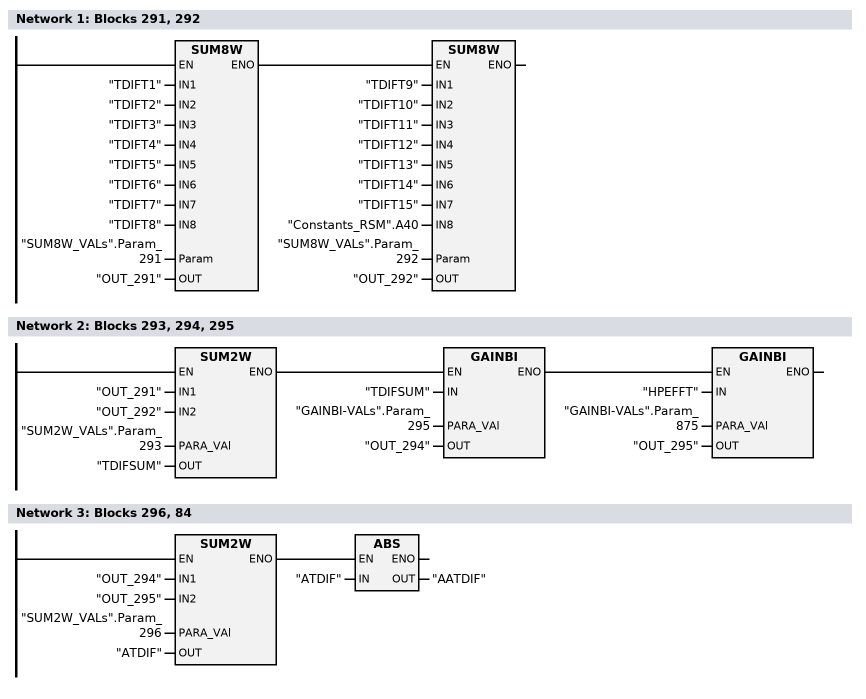
NETWORK
TITLE = Blocks 291, 292
      A(;
      CALL  "SUM8W" (
           IN1                      := "TDIFT1",
           IN2                      := "TDIFT2",
           IN3                      := "TDIFT3",
           IN4                      := "TDIFT4",
           IN5                      := "TDIFT5",
           IN6                      := "TDIFT6",
           IN7                      := "TDIFT7",
           IN8                      := "TDIFT8",
           Param                    := "SUM8W_VALs".Param_291,
           OUT                      := "OUT_291");
      A     BR;
      );
      JNB   _001;
      CALL  "SUM8W" (
           IN1                      := "TDIFT9",
           IN2                      := "TDIFT10",
           IN3                      := "TDIFT11",
           IN4                      := "TDIFT12",
           IN5                      := "TDIFT13",
           IN6                      := "TDIFT14",
           IN7                      := "TDIFT15",
           IN8                      := "Constants_RSM".A40,
           Param                    := "SUM8W_VALs".Param_292,
           OUT                      := "OUT_292");
_001: NOP   0;
NETWORK
TITLE = Blocks 293, 294, 295
      A(;
      A(;
      CALL  "SUM2W" (
           IN1                      := "OUT_291",
           IN2                      := "OUT_292",
           PARA_VAl                 := "SUM2W_VALs".Param_293,
           OUT                      := "TDIFSUM");
      A     BR;
      );
      JNB   _002;
      CALL  "GAINBI" (
           IN                       := "TDIFSUM",
           PARA_VAl                 := "GAINBI-VALs".Param_295,
           OUT                      := "OUT_294");
_002: A     BR;
      );
      JNB   _003;
      CALL  "GAINBI" (
           IN                       := "HPEFFT",
           PARA_VAl                 := "GAINBI-VALs".Param_875,
           OUT                      := "OUT_295");
_003: NOP   0;
NETWORK
TITLE = Blocks 296, 84
//IN1 of block 296 should be -ve as shown in sheet 16 (RSM)
      A(;
      CALL  "SUM2W" (
           IN1                      := "OUT_294",
           IN2                      := "OUT_295",
           PARA_VAl                 := "SUM2W_VALs".Param_296,
           OUT                      := "ATDIF");
      A     BR;
      );
      JNB   _004;
      L     "ATDIF";
      ABS;
      T     "AATDIF";
_004: NOP   0;
END_FUNCTION

FUNCTION "Sheet 17 (RSM)" : VOID	// FC 53
TITLE = Sheet 17 (RSM)
//% ROTOR STRESS LIMIT (Analog)
//Note: PV gain of all the XSUM blocks should be -ve as shown in sheet 17 (RSM).
AUTHOR : RJ
FAMILY : RSM
VERSION : 0.1
BEGIN
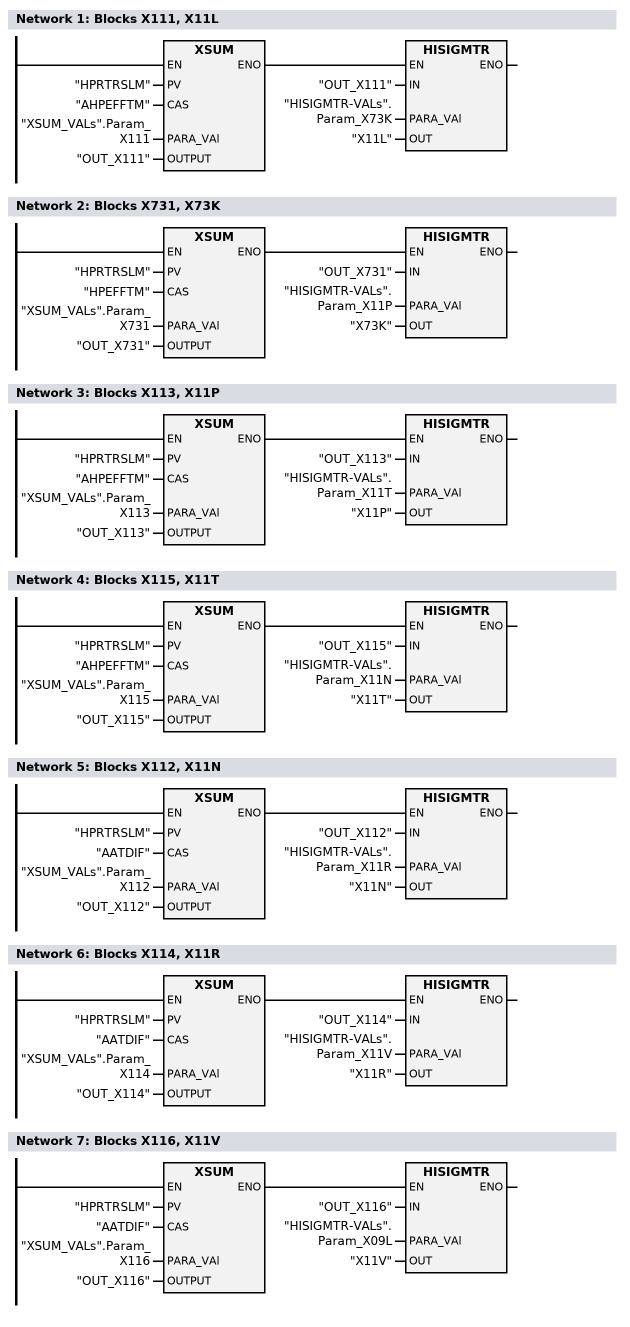
NETWORK
TITLE = Blocks X111, X11L
      A(;
      CALL  "XSUM" (
           PV                       := "HPRTRSLM",
           CAS                      := "AHPEFFTM",
           PARA_VAl                 := "XSUM_VALs".Param_X111,
           OUTPUT                   := "OUT_X111");
      A     BR;
      );
      JNB   _001;
      CALL  "HISIGMTR" (
           IN                       := "OUT_X111",
           PARA_VAl                 := "HISIGMTR-VALs".Param_X73K,
           OUT                      := "X11L");
_001: NOP   0;
NETWORK
TITLE = Blocks X731, X73K
      A(;
      CALL  "XSUM" (
           PV                       := "HPRTRSLM",
           CAS                      := "HPEFFTM",
           PARA_VAl                 := "XSUM_VALs".Param_X731,
           OUTPUT                   := "OUT_X731");
      A     BR;
      );
      JNB   _002;
      CALL  "HISIGMTR" (
           IN                       := "OUT_X731",
           PARA_VAl                 := "HISIGMTR-VALs".Param_X11P,
           OUT                      := "X73K");
_002: NOP   0;
NETWORK
TITLE = Blocks X113, X11P
      A(;
      CALL  "XSUM" (
           PV                       := "HPRTRSLM",
           CAS                      := "AHPEFFTM",
           PARA_VAl                 := "XSUM_VALs".Param_X113,
           OUTPUT                   := "OUT_X113");
      A     BR;
      );
      JNB   _003;
      CALL  "HISIGMTR" (
           IN                       := "OUT_X113",
           PARA_VAl                 := "HISIGMTR-VALs".Param_X11T,
           OUT                      := "X11P");
_003: NOP   0;
NETWORK
TITLE = Blocks X115, X11T
      A(;
      CALL  "XSUM" (
           PV                       := "HPRTRSLM",
           CAS                      := "AHPEFFTM",
           PARA_VAl                 := "XSUM_VALs".Param_X115,
           OUTPUT                   := "OUT_X115");
      A     BR;
      );
      JNB   _004;
      CALL  "HISIGMTR" (
           IN                       := "OUT_X115",
           PARA_VAl                 := "HISIGMTR-VALs".Param_X11N,
           OUT                      := "X11T");
_004: NOP   0;
NETWORK
TITLE = Blocks X112, X11N
      A(;
      CALL  "XSUM" (
           PV                       := "HPRTRSLM",
           CAS                      := "AATDIF",
           PARA_VAl                 := "XSUM_VALs".Param_X112,
           OUTPUT                   := "OUT_X112");
      A     BR;
      );
      JNB   _005;
      CALL  "HISIGMTR" (
           IN                       := "OUT_X112",
           PARA_VAl                 := "HISIGMTR-VALs".Param_X11R,
           OUT                      := "X11N");
_005: NOP   0;
NETWORK
TITLE = Blocks X114, X11R
      A(;
      CALL  "XSUM" (
           PV                       := "HPRTRSLM",
           CAS                      := "AATDIF",
           PARA_VAl                 := "XSUM_VALs".Param_X114,
           OUTPUT                   := "OUT_X114");
      A     BR;
      );
      JNB   _006;
      CALL  "HISIGMTR" (
           IN                       := "OUT_X114",
           PARA_VAl                 := "HISIGMTR-VALs".Param_X11V,
           OUT                      := "X11R");
_006: NOP   0;
NETWORK
TITLE = Blocks X116, X11V
      A(;
      CALL  "XSUM" (
           PV                       := "HPRTRSLM",
           CAS                      := "AATDIF",
           PARA_VAl                 := "XSUM_VALs".Param_X116,
           OUTPUT                   := "OUT_X116");
      A     BR;
      );
      JNB   _007;
      CALL  "HISIGMTR" (
           IN                       := "OUT_X116",
           PARA_VAl                 := "HISIGMTR-VALs".Param_X09L,
           OUT                      := "X11V");
_007: NOP   0;
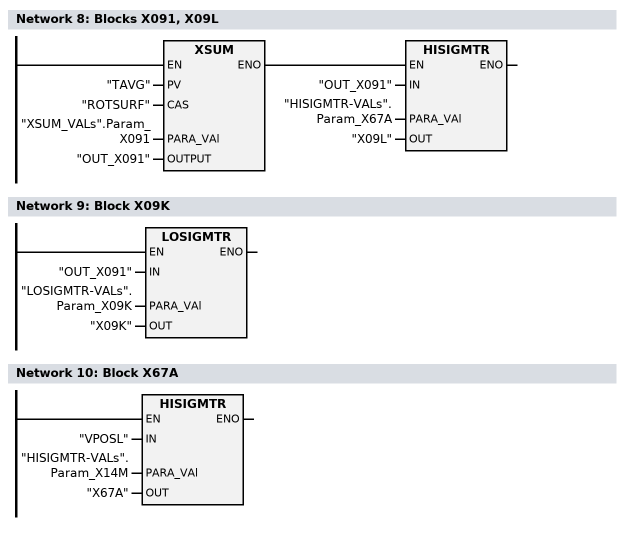
NETWORK
TITLE = Blocks X091, X09L
      A(;
      CALL  "XSUM" (
           PV                       := "TAVG",
           CAS                      := "ROTSURF",
           PARA_VAl                 := "XSUM_VALs".Param_X091,
           OUTPUT                   := "OUT_X091");
      A     BR;
      );
      JNB   _008;
      CALL  "HISIGMTR" (
           IN                       := "OUT_X091",
           PARA_VAl                 := "HISIGMTR-VALs".Param_X67A,
           OUT                      := "X09L");
_008: NOP   0;
NETWORK
TITLE = Block X09K
      CALL  "LOSIGMTR" (
           IN                       := "OUT_X091",
           PARA_VAl                 := "LOSIGMTR-VALs".Param_X09K,
           OUT                      := "X09K");
      NOP   0;
NETWORK
TITLE = Block X67A
      CALL  "HISIGMTR" (
           IN                       := "VPOSL",
           PARA_VAl                 := "HISIGMTR-VALs".Param_X14M,
           OUT                      := "X67A");
      NOP   0;
END_FUNCTION

FUNCTION "XMULT" : VOID	// FC 54
AUTHOR : RJ
VERSION : 0.0
VAR_INPUT
  PV : REAL ;
  CAS : REAL ;
  Param : STRUCT
   PV_GAIN : REAL ;
   PV_BIAS : REAL ;
   CAS_GAIN : REAL ;
   CAS_BIAS : REAL ;
   SCALE_TOP : REAL ;
   SCALE_BOT : REAL ;
  END_STRUCT ;
END_VAR
VAR_OUTPUT
  OUT : REAL ;
END_VAR
VAR_TEMP
  PVGB : REAL ;
  CASGB : REAL ;
END_VAR
BEGIN
// body was compiled from an SCL source; compiled code not shown
END_FUNCTION

FUNCTION "Sheet 18 (RSM)" : VOID	// FC 55
TITLE = Sheet 18 (RSM)
//SMW INC/DEC (Analog)
AUTHOR : RJ
FAMILY : RSM
VERSION : 0.1
BEGIN
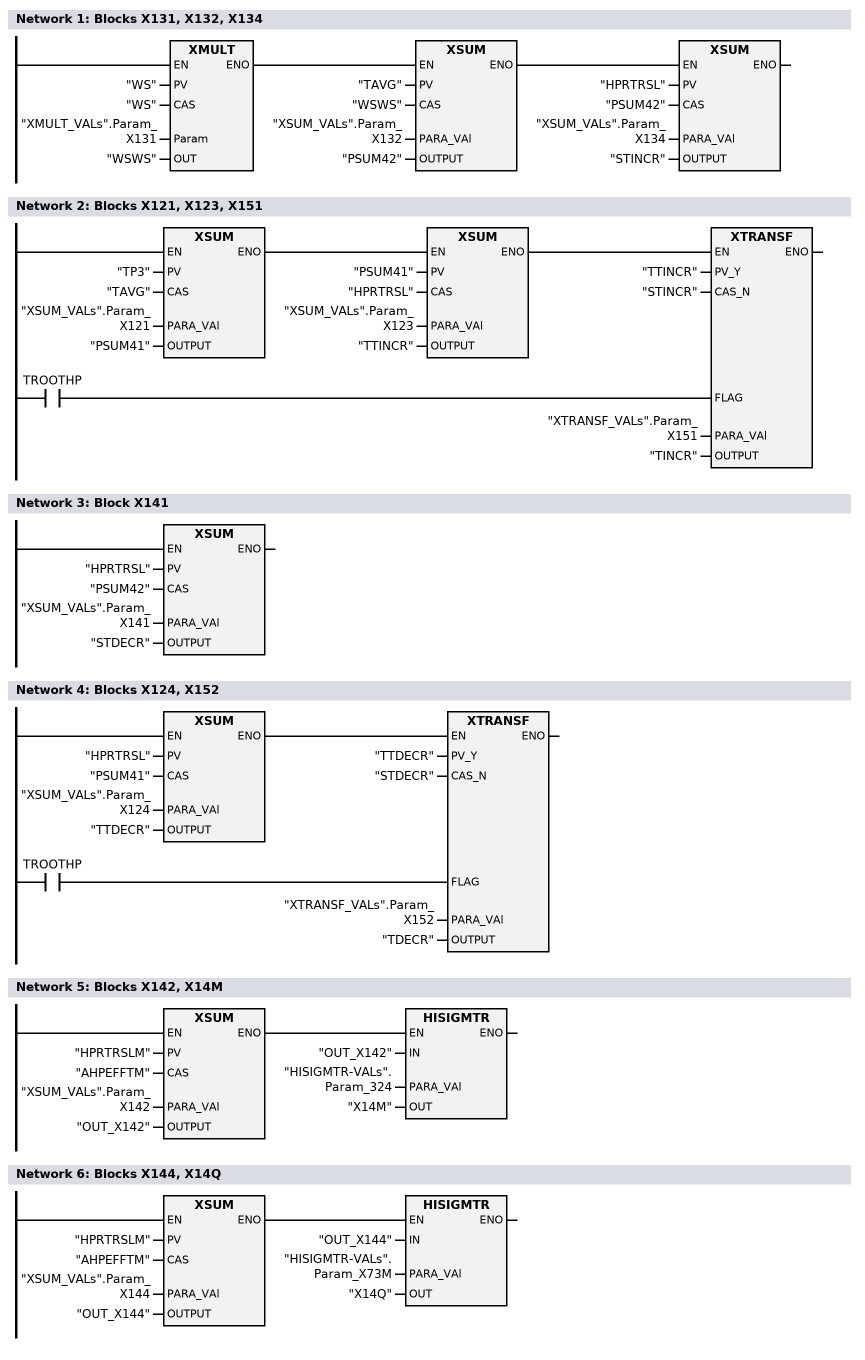
NETWORK
TITLE = Blocks X131, X132, X134
      A(;
      A(;
      CALL  "XMULT" (
           PV                       := "WS",
           CAS                      := "WS",
           Param                    := "XMULT_VALs".Param_X131,
           OUT                      := "WSWS");
      A     BR;
      );
      JNB   _001;
      CALL  "XSUM" (
           PV                       := "TAVG",
           CAS                      := "WSWS",
           PARA_VAl                 := "XSUM_VALs".Param_X132,
           OUTPUT                   := "PSUM42");
_001: A     BR;
      );
      JNB   _002;
      CALL  "XSUM" (
           PV                       := "HPRTRSL",
           CAS                      := "PSUM42",
           PARA_VAl                 := "XSUM_VALs".Param_X134,
           OUTPUT                   := "STINCR");
_002: NOP   0;
NETWORK
TITLE = Blocks X121, X123, X151
      A     "TROOTHP";
      =     L 0.0;
      BLD   103;
      A(;
      A(;
      CALL  "XSUM" (
           PV                       := "TP3",
           CAS                      := "TAVG",
           PARA_VAl                 := "XSUM_VALs".Param_X121,
           OUTPUT                   := "PSUM41");
      A     BR;
      );
      JNB   _003;
      CALL  "XSUM" (
           PV                       := "PSUM41",
           CAS                      := "HPRTRSL",
           PARA_VAl                 := "XSUM_VALs".Param_X123,
           OUTPUT                   := "TTINCR");
_003: A     BR;
      );
      JNB   _004;
      CALL  "XTRANSF" (
           PV_Y                     := "TTINCR",
           CAS_N                    := "STINCR",
           FLAG                     := L 0.0,
           PARA_VAl                 := "XTRANSF_VALs".Param_X151,
           OUTPUT                   := "TINCR");
_004: NOP   0;
NETWORK
TITLE = Block X141
//PV gain of the block should be -ve as shown in sheet 18 (RSM)
      CALL  "XSUM" (
           PV                       := "HPRTRSL",
           CAS                      := "PSUM42",
           PARA_VAl                 := "XSUM_VALs".Param_X141,
           OUTPUT                   := "STDECR");
      NOP   0;
NETWORK
TITLE = Blocks X124, X152
//PV gain of the block X124 should be -ve as shown in sheet 18 (RSM)
      A     "TROOTHP";
      =     L 0.0;
      BLD   103;
      A(;
      CALL  "XSUM" (
           PV                       := "HPRTRSL",
           CAS                      := "PSUM41",
           PARA_VAl                 := "XSUM_VALs".Param_X124,
           OUTPUT                   := "TTDECR");
      A     BR;
      );
      JNB   _005;
      CALL  "XTRANSF" (
           PV_Y                     := "TTDECR",
           CAS_N                    := "STDECR",
           FLAG                     := L 0.0,
           PARA_VAl                 := "XTRANSF_VALs".Param_X152,
           OUTPUT                   := "TDECR");
_005: NOP   0;
NETWORK
TITLE = Blocks X142, X14M
//PV gain of the block X142 should be -ve as shown in sheet 18 (RSM)
      A(;
      CALL  "XSUM" (
           PV                       := "HPRTRSLM",
           CAS                      := "AHPEFFTM",
           PARA_VAl                 := "XSUM_VALs".Param_X142,
           OUTPUT                   := "OUT_X142");
      A     BR;
      );
      JNB   _006;
      CALL  "HISIGMTR" (
           IN                       := "OUT_X142",
           PARA_VAl                 := "HISIGMTR-VALs".Param_324,
           OUT                      := "X14M");
_006: NOP   0;
NETWORK
TITLE = Blocks X144, X14Q
//PV gain of the block X144 should be -ve as shown in sheet 18 (RSM)
      A(;
      CALL  "XSUM" (
           PV                       := "HPRTRSLM",
           CAS                      := "AHPEFFTM",
           PARA_VAl                 := "XSUM_VALs".Param_X144,
           OUTPUT                   := "OUT_X144");
      A     BR;
      );
      JNB   _007;
      CALL  "HISIGMTR" (
           IN                       := "OUT_X144",
           PARA_VAl                 := "HISIGMTR-VALs".Param_X73M,
           OUT                      := "X14Q");
_007: NOP   0;
END_FUNCTION

FUNCTION "Sheet 19 (RSM)" : VOID	// FC 57
TITLE = Sheet 19 (RSM)
//TBP (Analog)
AUTHOR : RJ
FAMILY : RSM
VERSION : 0.1
BEGIN
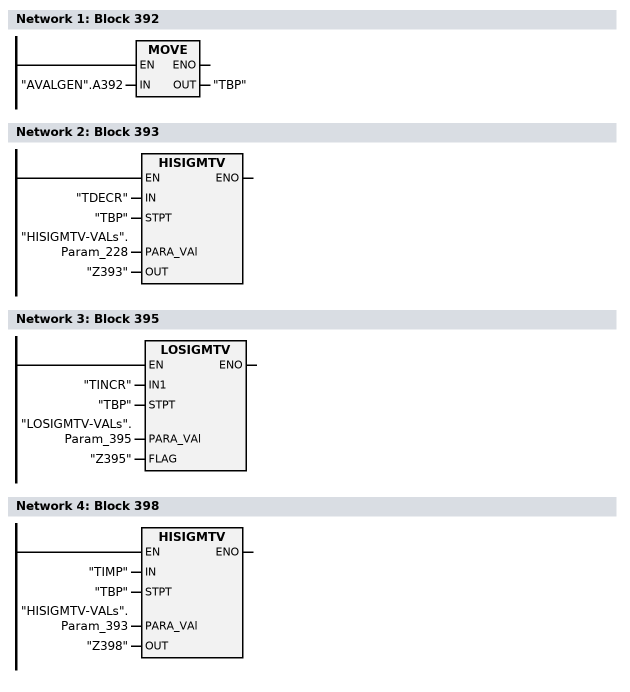
NETWORK
TITLE = Block 392
      L     "AVALGEN".A392;
      T     "TBP";
      NOP   0;
NETWORK
TITLE = Block 393
      CALL  "HISIGMTV" (
           IN                       := "TDECR",
           STPT                     := "TBP",
           PARA_VAl                 := "HISIGMTV-VALs".Param_228,
           OUT                      := "Z393");
      NOP   0;
NETWORK
TITLE = Block 395
      CALL  "LOSIGMTV" (
           IN1                      := "TINCR",
           STPT                     := "TBP",
           PARA_VAl                 := "LOSIGMTV-VALs".Param_395,
           FLAG                     := "Z395");
      NOP   0;
NETWORK
TITLE = Block 398
      CALL  "HISIGMTV" (
           IN                       := "TIMP",
           STPT                     := "TBP",
           PARA_VAl                 := "HISIGMTV-VALs".Param_393,
           OUT                      := "Z398");
      NOP   0;
END_FUNCTION

FUNCTION "Sheet 20 (RSM)" : VOID	// FC 58
TITLE = Sheet 20 (RSM)
//MWINCR (Analog)
AUTHOR : RJ
FAMILY : RSM
VERSION : 0.1
BEGIN
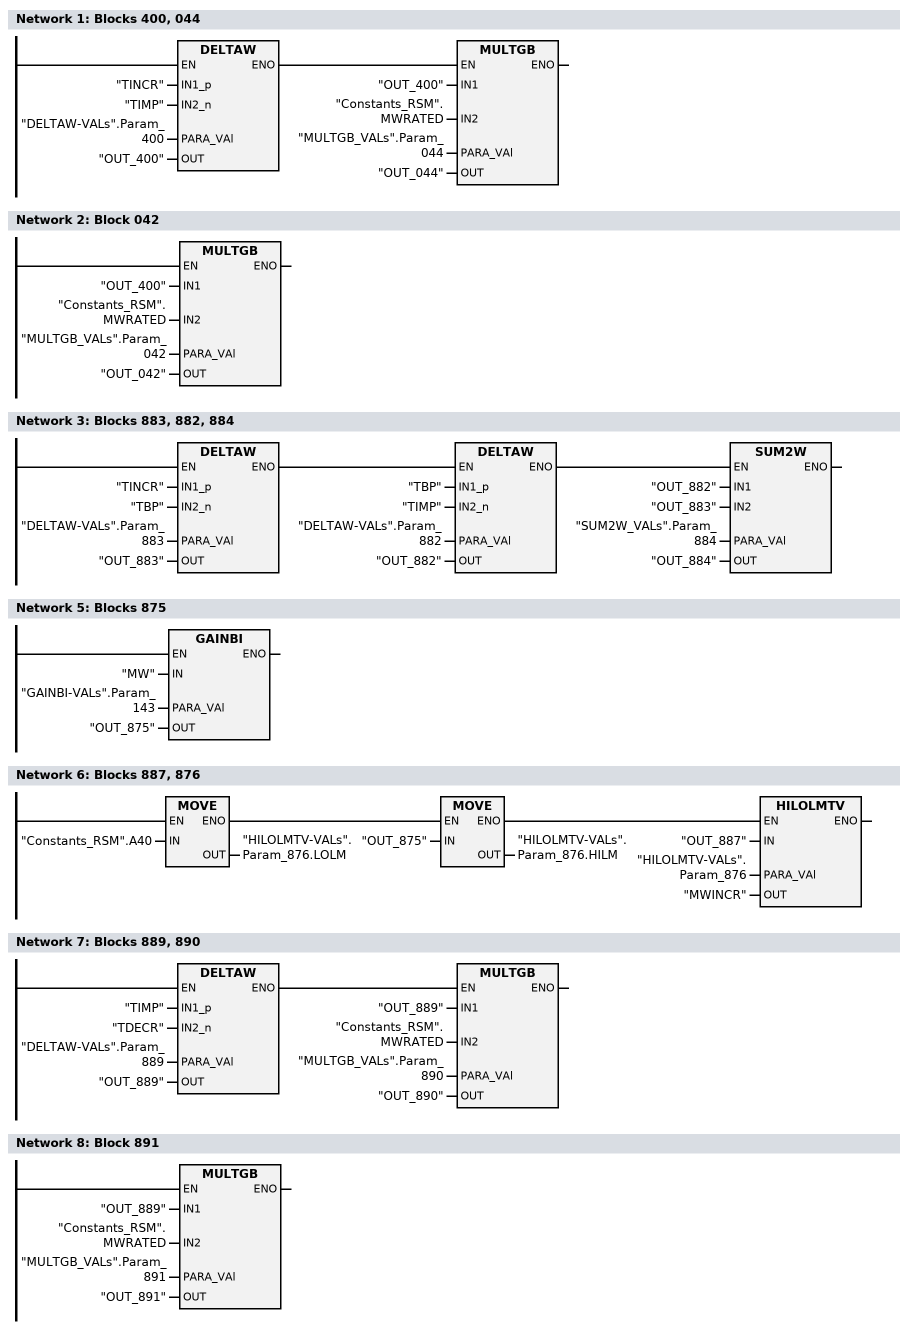
NETWORK
TITLE = Blocks 400, 044
      A(;
      CALL  "DELTAW" (
           IN1_p                    := "TINCR",
           IN2_n                    := "TIMP",
           PARA_VAl                 := "DELTAW-VALs".Param_400,
           OUT                      := "OUT_400");
      A     BR;
      );
      JNB   _001;
      CALL  "MULTGB" (
           IN1                      := "OUT_400",
           IN2                      := "Constants_RSM".MWRATED,
           PARA_VAl                 := "MULTGB_VALs".Param_044,
           OUT                      := "OUT_044");
_001: NOP   0;
NETWORK
TITLE = Block 042
      CALL  "MULTGB" (
           IN1                      := "OUT_400",
           IN2                      := "Constants_RSM".MWRATED,
           PARA_VAl                 := "MULTGB_VALs".Param_042,
           OUT                      := "OUT_042");
      NOP   0;
NETWORK
TITLE = Blocks 883, 882, 884
      A(;
      A(;
      CALL  "DELTAW" (
           IN1_p                    := "TINCR",
           IN2_n                    := "TBP",
           PARA_VAl                 := "DELTAW-VALs".Param_883,
           OUT                      := "OUT_883");
      A     BR;
      );
      JNB   _002;
      CALL  "DELTAW" (
           IN1_p                    := "TBP",
           IN2_n                    := "TIMP",
           PARA_VAl                 := "DELTAW-VALs".Param_882,
           OUT                      := "OUT_882");
_002: A     BR;
      );
      JNB   _003;
      CALL  "SUM2W" (
           IN1                      := "OUT_882",
           IN2                      := "OUT_883",
           PARA_VAl                 := "SUM2W_VALs".Param_884,
           OUT                      := "OUT_884");
_003: NOP   0;
NETWORK
TITLE = Blocks 885, 886
      A     "Z745";
      =     L 0.0;
      BLD   103;
      A(;
      A     "Z395";
      =     L 0.1;
      BLD   103;
      A(;
      CALL  "MULTGB" (
           IN1                      := "OUT_884",
           IN2                      := "Constants_RSM".MWRATED,
           PARA_VAl                 := "MULTGB_VALs".Param_885,
           OUT                      := "OUT_885");
      A     BR;
      );
      JNB   _004;
      CALL  "TRANSF" (
           FLAG                     := L 0.1,
           IN1_y                    := "OUT_044",
           IN2_n                    := "OUT_885",
           OUT                      := "OUT_886");
_004: A     BR;
      );
      JNB   _005;
      CALL  "TRANSF" (
           FLAG                     := L 0.0,
           IN1_y                    := "OUT_042",
           IN2_n                    := "OUT_886",
           OUT                      := "OUT_887");
_005: NOP   0;
NETWORK
TITLE = Blocks 875
      CALL  "GAINBI" (
           IN                       := "MW",
           PARA_VAl                 := "GAINBI-VALs".Param_143,
           OUT                      := "OUT_875");
      NOP   0;
NETWORK
TITLE = Blocks 887, 876
      A(;
      A(;
      L     "Constants_RSM".A40;
      T     "HILOLMTV-VALs".Param_876.LOLM;
      SET;
      SAVE;
      CLR;
      A     BR;
      );
      JNB   _006;
      L     "OUT_875";
      T     "HILOLMTV-VALs".Param_876.HILM;
      SET;
      SAVE;
      CLR;
_006: A     BR;
      );
      JNB   _007;
      CALL  "HILOLMTV" (
           IN                       := "OUT_887",
           PARA_VAl                 := "HILOLMTV-VALs".Param_876,
           OUT                      := "MWINCR");
_007: NOP   0;
NETWORK
TITLE = Blocks 889, 890
      A(;
      CALL  "DELTAW" (
           IN1_p                    := "TIMP",
           IN2_n                    := "TDECR",
           PARA_VAl                 := "DELTAW-VALs".Param_889,
           OUT                      := "OUT_889");
      A     BR;
      );
      JNB   _008;
      CALL  "MULTGB" (
           IN1                      := "OUT_889",
           IN2                      := "Constants_RSM".MWRATED,
           PARA_VAl                 := "MULTGB_VALs".Param_890,
           OUT                      := "OUT_890");
_008: NOP   0;
NETWORK
TITLE = Block 891
      CALL  "MULTGB" (
           IN1                      := "OUT_889",
           IN2                      := "Constants_RSM".MWRATED,
           PARA_VAl                 := "MULTGB_VALs".Param_891,
           OUT                      := "OUT_891");
      NOP   0;
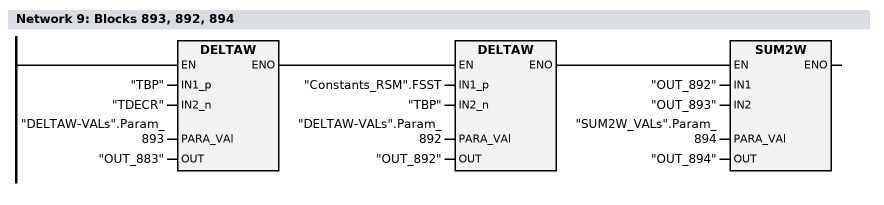
NETWORK
TITLE = Blocks 893, 892, 894
      A(;
      A(;
      CALL  "DELTAW" (
           IN1_p                    := "TBP",
           IN2_n                    := "TDECR",
           PARA_VAl                 := "DELTAW-VALs".Param_893,
           OUT                      := "OUT_883");
      A     BR;
      );
      JNB   _009;
      CALL  "DELTAW" (
           IN1_p                    := "Constants_RSM".FSST,
           IN2_n                    := "TBP",
           PARA_VAl                 := "DELTAW-VALs".Param_892,
           OUT                      := "OUT_892");
_009: A     BR;
      );
      JNB   _00a;
      CALL  "SUM2W" (
           IN1                      := "OUT_892",
           IN2                      := "OUT_893",
           PARA_VAl                 := "SUM2W_VALs".Param_894,
           OUT                      := "OUT_894");
_00a: NOP   0;
NETWORK
TITLE = Blocks 895, 896, 897
      A     "Z393";
      =     L 0.0;
      BLD   103;
      A(;
      A     "Z747";
      =     L 0.1;
      BLD   103;
      A(;
      CALL  "MULTGB" (
           IN1                      := "OUT_894",
           IN2                      := "Constants_RSM".MWRATED,
           PARA_VAl                 := "MULTGB_VALs".Param_895,
           OUT                      := "OUT_895");
      A     BR;
      );
      JNB   _00b;
      CALL  "TRANSF" (
           FLAG                     := L 0.1,
           IN1_y                    := "OUT_890",
           IN2_n                    := "OUT_895",
           OUT                      := "OUT_896");
_00b: A     BR;
      );
      JNB   _00c;
      CALL  "TRANSF" (
           FLAG                     := L 0.0,
           IN1_y                    := "OUT_891",
           IN2_n                    := "OUT_896",
           OUT                      := "OUT_897");
_00c: NOP   0;
END_FUNCTION

FUNCTION "Sheet 21 (RSM)" : VOID	// FC 59
TITLE = Sheet 21 (RSM)
//ATC RATE & LOAD RESERVE (Analog)
AUTHOR : RJ
FAMILY : RSM
VERSION : 0.1
BEGIN
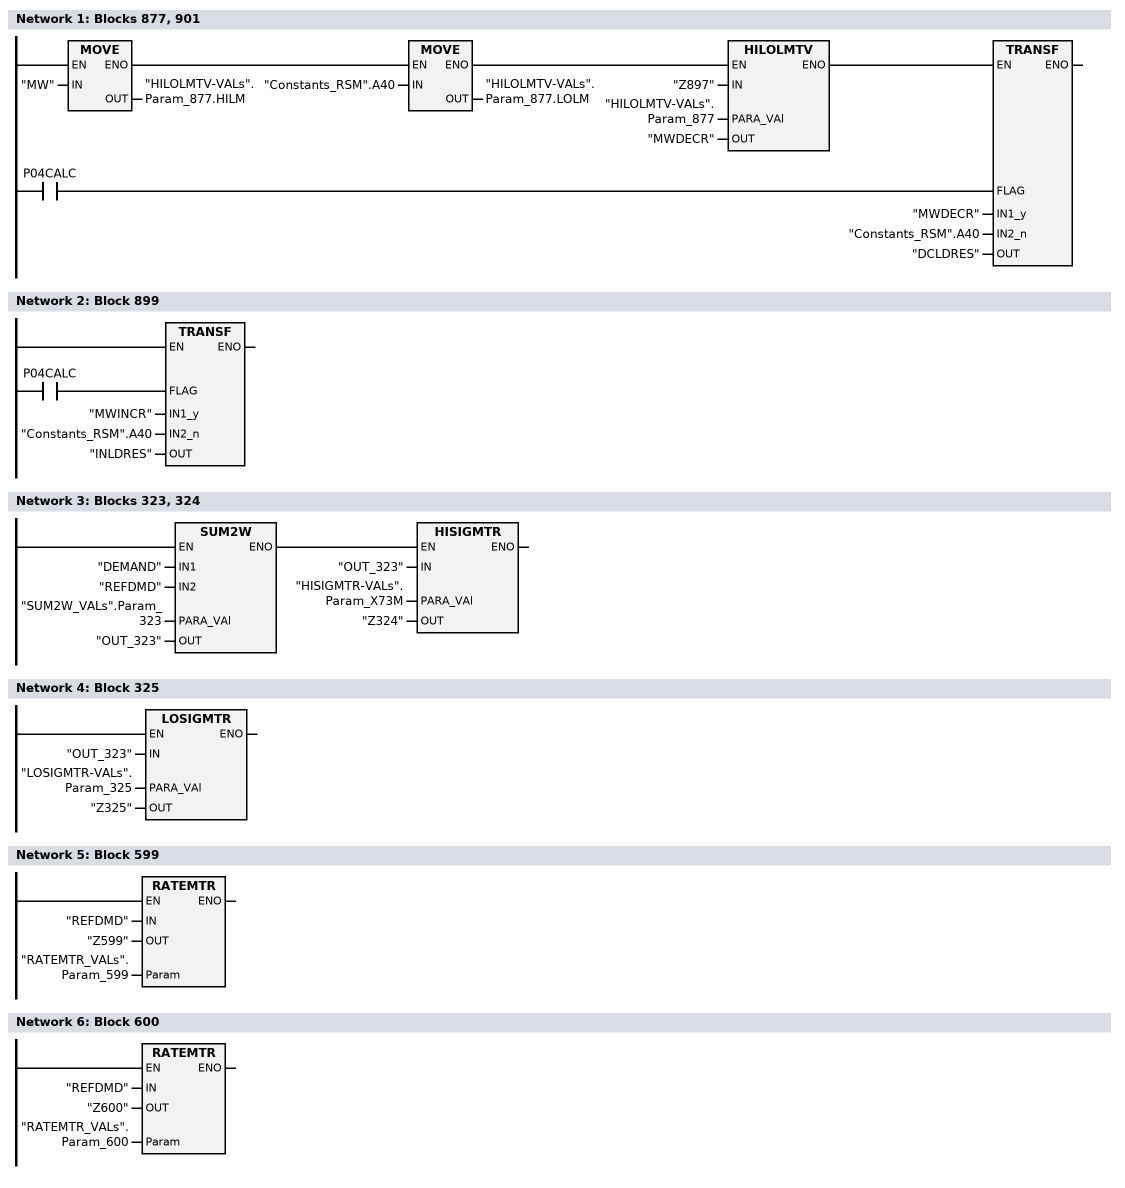
NETWORK
TITLE = Blocks 877, 901
      A     "P04CALC";
      =     L 0.0;
      BLD   103;
      A(;
      A(;
      A(;
      L     "MW";
      T     "HILOLMTV-VALs".Param_877.HILM;
      SET;
      SAVE;
      CLR;
      A     BR;
      );
      JNB   _001;
      L     "Constants_RSM".A40;
      T     "HILOLMTV-VALs".Param_877.LOLM;
      SET;
      SAVE;
      CLR;
_001: A     BR;
      );
      JNB   _002;
      CALL  "HILOLMTV" (
           IN                       := "Z897",
           PARA_VAl                 := "HILOLMTV-VALs".Param_877,
           OUT                      := "MWDECR");
_002: A     BR;
      );
      JNB   _003;
      CALL  "TRANSF" (
           FLAG                     := L 0.0,
           IN1_y                    := "MWDECR",
           IN2_n                    := "Constants_RSM".A40,
           OUT                      := "DCLDRES");
_003: NOP   0;
NETWORK
TITLE = Block 899
      A     "P04CALC";
      =     L 0.0;
      BLD   103;
      CALL  "TRANSF" (
           FLAG                     := L 0.0,
           IN1_y                    := "MWINCR",
           IN2_n                    := "Constants_RSM".A40,
           OUT                      := "INLDRES");
      NOP   0;
NETWORK
TITLE = Blocks 323, 324
//IN2 of the block 323 should have a -ve weight as shown in sheet 21 (RSM).
      A(;
      CALL  "SUM2W" (
           IN1                      := "DEMAND",
           IN2                      := "REFDMD",
           PARA_VAl                 := "SUM2W_VALs".Param_323,
           OUT                      := "OUT_323");
      A     BR;
      );
      JNB   _004;
      CALL  "HISIGMTR" (
           IN                       := "OUT_323",
           PARA_VAl                 := "HISIGMTR-VALs".Param_X73M,
           OUT                      := "Z324");
_004: NOP   0;
NETWORK
TITLE = Block 325
      CALL  "LOSIGMTR" (
           IN                       := "OUT_323",
           PARA_VAl                 := "LOSIGMTR-VALs".Param_325,
           OUT                      := "Z325");
      NOP   0;
NETWORK
TITLE = Block 599
      CALL  "RATEMTR" (
           IN                       := "REFDMD",
           OUT                      := "Z599",
           Param                    := "RATEMTR_VALs".Param_599);
      NOP   0;
NETWORK
TITLE = Block 600
      CALL  "RATEMTR" (
           IN                       := "REFDMD",
           OUT                      := "Z600",
           Param                    := "RATEMTR_VALs".Param_600);
      NOP   0;
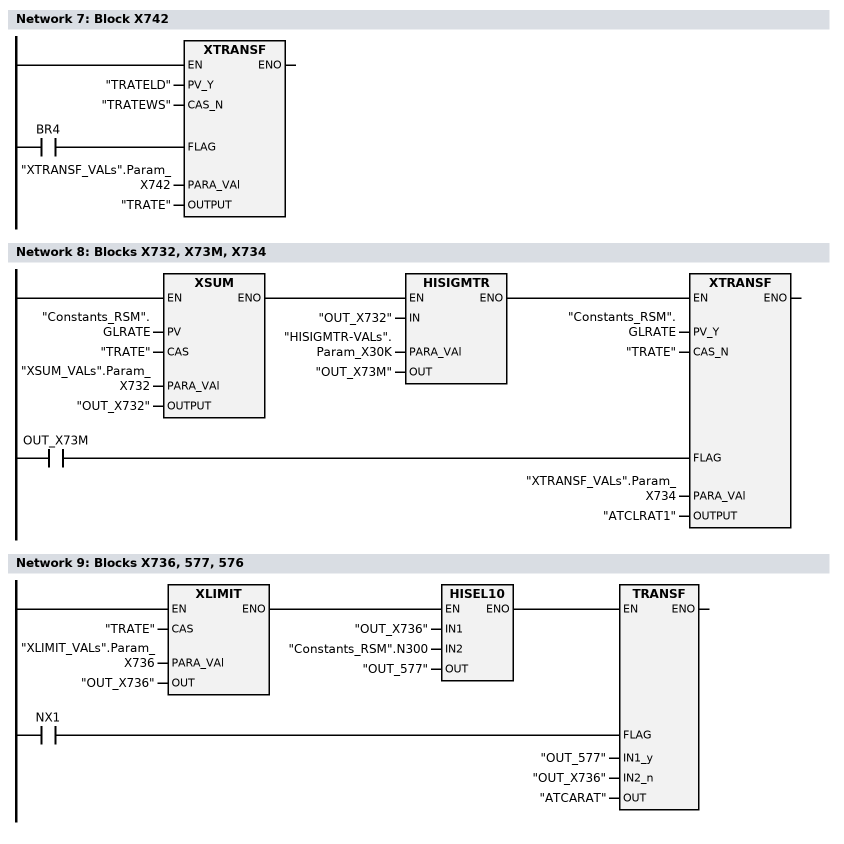
NETWORK
TITLE = Block X742
      A     "BR4";
      =     L 0.0;
      BLD   103;
      CALL  "XTRANSF" (
           PV_Y                     := "TRATELD",
           CAS_N                    := "TRATEWS",
           FLAG                     := L 0.0,
           PARA_VAl                 := "XTRANSF_VALs".Param_X742,
           OUTPUT                   := "TRATE");
      NOP   0;
NETWORK
TITLE = Blocks X732, X73M, X734
//PV input of the block X732 should have -ve weight as shown in sheet 21 (RSM).
      A     "OUT_X73M";
      =     L 0.0;
      BLD   103;
      A(;
      A(;
      CALL  "XSUM" (
           PV                       := "Constants_RSM".GLRATE,
           CAS                      := "TRATE",
           PARA_VAl                 := "XSUM_VALs".Param_X732,
           OUTPUT                   := "OUT_X732");
      A     BR;
      );
      JNB   _005;
      CALL  "HISIGMTR" (
           IN                       := "OUT_X732",
           PARA_VAl                 := "HISIGMTR-VALs".Param_X30K,
           OUT                      := "OUT_X73M");
_005: A     BR;
      );
      JNB   _006;
      CALL  "XTRANSF" (
           PV_Y                     := "Constants_RSM".GLRATE,
           CAS_N                    := "TRATE",
           FLAG                     := L 0.0,
           PARA_VAl                 := "XTRANSF_VALs".Param_X734,
           OUTPUT                   := "ATCLRAT1");
_006: NOP   0;
NETWORK
TITLE = Blocks X736, 577, 576
      A     "NX1";
      =     L 0.0;
      BLD   103;
      A(;
      A(;
      CALL  "XLIMIT" (
           CAS                      := "TRATE",
           PARA_VAl                 := "XLIMIT_VALs".Param_X736,
           OUT                      := "OUT_X736");
      A     BR;
      );
      JNB   _007;
      CALL  "HISEL10" (
           IN1                      := "OUT_X736",
           IN2                      := "Constants_RSM".N300,
           OUT                      := "OUT_577");
_007: A     BR;
      );
      JNB   _008;
      CALL  "TRANSF" (
           FLAG                     := L 0.0,
           IN1_y                    := "OUT_577",
           IN2_n                    := "OUT_X736",
           OUT                      := "ATCARAT");
_008: NOP   0;
END_FUNCTION

FUNCTION "SUM4W" : VOID	// FC 60
AUTHOR : Sabeeh
VERSION : 0.0
VAR_INPUT
  IN1 : REAL ;
  IN2 : REAL ;
  IN3 : REAL ;
  IN4 : REAL ;
  PARA_VAl : STRUCT
   WT1 : REAL ;
   WT2 : REAL ;
   WT3 : REAL ;
   WT4 : REAL ;
  END_STRUCT ;
END_VAR
VAR_OUTPUT
  OUT : REAL ;
END_VAR
BEGIN
// body was compiled from an SCL source; compiled code not shown
END_FUNCTION

FUNCTION "Sheet 22 (RSM)" : VOID	// FC 61
TITLE = Sheet 22 (RSM)
//REQ. STM CHEST METAL TEMP (Analog)
AUTHOR : RJ
FAMILY : RSM
VERSION : 0.1
BEGIN
NETWORK
TITLE = Blocks 159, 144
      A(;
      A     "BR4";
      =     L 0.0;
      BLD   103;
      CALL  "TRANSF" (
           FLAG                     := L 0.0,
           IN1_y                    := "Constants_RSM".NDIFLM,
           IN2_n                    := "Constants_RSM".HOTDIFLM,
           OUT                      := "OUT_159");
      A     BR;
      );
      JNB   _001;
      CALL  "GAINBI" (
           IN                       := "OUT_159",
           PARA_VAl                 := "GAINBI-VALs".Param_144,
           OUT                      := "HPRSLNEG");
_001: NOP   0;
